LIN {X -0.181,Y -423.793,Z 1219.594,A 0.000,B 0.000,C 90.000,E1 286.913} C_DIS
LIN {X -0.003,Y -430.915,Z 1219.589,A 0.000,B 0.000,C 90.000,E1 286.079} C_DIS
LIN {X -0.077,Y -435.410,Z 1219.586,A 0.000,B 0.000,C 90.000,E1 285.552} C_DIS
LIN {X 0.192,Y -441.538,Z 1219.582,A 0.000,B 0.000,C 90.000,E1 284.717} C_DIS
LIN {X 0.092,Y -447.112,Z 1219.578,A 0.000,B 0.000,C 90.000,E1 283.939} C_DIS
LIN {X -0.076,Y -452.101,Z 1219.573,A 0.000,B 0.000,C 90.000,E1 283.175} C_DIS
LIN {X 0.247,Y -456.380,Z 1219.569,A 0.000,B 0.000,C 90.000,E1 282.355} C_DIS
LIN {X 0.160,Y -459.934,Z 1219.564,A 0.000,B 0.000,C 90.000,E1 281.591} C_DIS
LIN {X 0.182,Y -461.942,Z 1219.562,A 0.000,B 0.000,C 90.000,E1 281.074} C_DIS
LIN {X -0.154,Y -463.736,Z 1219.559,A 0.000,B 0.000,C 90.000,E1 280.602} C_DIS
LIN {X -0.028,Y -465.195,Z 1219.556,A 0.000,B 0.000,C 90.000,E1 280.074} C_DIS
LIN {X 0.030,Y -466.423,Z 1219.553,A 0.000,B 0.000,C 90.000,E1 279.557} C_DIS
LIN {X 0.174,Y -467.373,Z 1219.550,A 0.000,B 0.000,C 90.000,E1 279.029} C_DIS
LIN {X -0.212,Y -468.042,Z 1219.547,A 0.000,B 0.000,C 90.000,E1 278.568} C_DIS
LIN {X -0.128,Y -468.455,Z 1219.545,A 0.000,B 0.000,C 90.000,E1 278.049} C_DIS
LIN {X -0.038,Y -468.559,Z 1219.542,A 0.000,B 0.000,C 90.000,E1 277.530} C_DIS
LIN {X 0.114,Y -468.268,Z 1219.539,A 0.000,B 0.000,C 90.000,E1 277.004} C_DIS
LIN {X 0.206,Y -467.592,Z 1219.536,A 0.000,B 0.000,C 90.000,E1 276.486} C_DIS
LIN {X -0.168,Y -466.535,Z 1219.533,A 0.000,B 0.000,C 90.000,E1 276.024} C_DIS
LIN {X -0.127,Y -465.025,Z 1219.531,A 0.000,B 0.000,C 90.000,E1 275.511} C_DIS
LIN {X 0.240,Y -461.969,Z 1219.526,A 0.000,B 0.000,C 90.000,E1 274.702} C_DIS
LIN {X -0.194,Y -459.223,Z 1219.523,A 0.000,B 0.000,C 90.000,E1 274.245} C_DIS
LIN {X -0.149,Y -455.714,Z 1219.521,A 0.000,B 0.000,C 90.000,E1 273.726} C_DIS
LIN {X -0.151,Y -451.325,Z 1219.518,A 0.000,B 0.000,C 90.000,E1 273.212} C_DIS
LIN {X -0.063,Y -445.903,Z 1219.515,A 0.000,B 0.000,C 90.000,E1 272.694} C_DIS
LIN {X -0.214,Y -442.714,Z 1219.514,A 0.000,B 0.000,C 90.000,E1 272.465} C_DIS
LIN {X 0.026,Y -436.059,Z 1219.511,A 0.000,B 0.000,C 90.000,E1 272.007} C_DIS
LIN {X -0.048,Y -428.864,Z 1219.509,A 0.000,B 0.000,C 90.000,E1 271.661} C_DIS
LIN {X -0.016,Y -421.713,Z 1219.508,A 0.000,B 0.000,C 90.000,E1 271.375} C_DIS
LIN {X 0.042,Y -411.638,Z 1219.506,A 0.000,B 0.000,C 90.000,E1 271.031} C_DIS
LIN {X 0.082,Y -401.252,Z 1219.504,A 0.000,B 0.000,C 90.000,E1 270.745} C_DIS
LIN {X 0.155,Y -394.190,Z 1219.503,A 0.000,B 0.000,C 90.000,E1 270.573} C_DIS
LIN {X -0.024,Y -385.825,Z 1219.503,A 0.000,B 0.000,C 90.000,E1 270.458} C_DIS
LIN {X 0.033,Y -376.005,Z 1219.502,A 0.000,B 0.000,C 90.000,E1 270.344} C_DIS
LIN {X 0.010,Y -364.057,Z 1219.502,A 0.000,B 0.000,C 90.000,E1 270.286} C_DIS
LIN {X -0.027,Y -181.581,Z 1219.502,A 0.000,B 0.000,C 90.000,E1 270.286} C_DIS
LIN {X -0.048,Y -180.830,Z 1219.472,A 0.000,B 0.000,C 90.000,E1 264.894} C_DIS
LIN {X 0.032,Y -178.936,Z 1219.443,A 0.000,B 0.000,C 90.000,E1 259.803} C_DIS
LIN {X -0.100,Y -175.984,Z 1219.415,A 0.000,B 0.000,C 90.000,E1 254.755} C_DIS
LIN {X 0.015,Y -175.481,Z 1219.410,A 0.000,B 0.000,C 90.000,E1 253.866} C_DIS
LIN {X 0.072,Y -172.227,Z 1219.387,A 0.000,B 0.000,C 90.000,E1 249.571} C_DIS
LIN {X 0.049,Y -171.704,Z 1219.382,A 0.000,B 0.000,C 90.000,E1 248.720} C_DIS
LIN {X -0.026,Y -167.298,Z 1219.353,A 0.000,B 0.000,C 90.000,E1 243.563} C_DIS
LIN {X 0.056,Y -166.676,Z 1219.348,A 0.000,B 0.000,C 90.000,E1 242.666} C_DIS
LIN {X -0.029,Y -162.658,Z 1219.324,A 0.000,B 0.000,C 90.000,E1 238.329} C_DIS
LIN {X 0.033,Y -161.347,Z 1219.314,A 0.000,B 0.000,C 90.000,E1 236.548} C_DIS
LIN {X 0.076,Y -157.341,Z 1219.290,A 0.000,B 0.000,C 90.000,E1 232.110} C_DIS
LIN {X 0.008,Y -155.327,Z 1219.275,A 0.000,B 0.000,C 90.000,E1 229.461} C_DIS
LIN {X -0.062,Y -151.679,Z 1219.250,A 0.000,B 0.000,C 90.000,E1 225.000} C_DIS
LIN {X -0.014,Y -150.543,Z 1219.240,A 0.000,B 0.000,C 90.000,E1 223.176} C_DIS
LIN {X 0.020,Y -147.269,Z 1219.215,A 0.000,B 0.000,C 90.000,E1 218.624} C_DIS
LIN {X -0.007,Y -145.296,Z 1219.194,A 0.000,B 0.000,C 90.000,E1 214.978} C_DIS
LIN {X -0.015,Y -142.392,Z 1219.164,A 0.000,B 0.000,C 90.000,E1 209.461} C_DIS
LIN {X 0.031,Y -141.372,Z 1219.148,A 0.000,B 0.000,C 90.000,E1 206.668} C_DIS
LIN {X 0.009,Y -139.346,Z 1219.112,A 0.000,B 0.000,C 90.000,E1 200.174} C_DIS
LIN {X 0.014,Y -139.018,Z 1219.102,A 0.000,B 0.000,C 90.000,E1 198.308} C_DIS
LIN {X 0.010,Y -138.343,Z 1219.055,A 0.000,B 0.000,C 90.000,E1 189.905} C_DIS
LIN {X 0.030,Y -139.392,Z 1219.008,A 0.000,B 0.000,C 90.000,E1 181.489} C_DIS
LIN {X -0.057,Y -141.291,Z 1218.972,A 0.000,B 0.000,C 90.000,E1 175.008} C_DIS
LIN {X 0.042,Y -142.654,Z 1218.957,A 0.000,B 0.000,C 90.000,E1 172.186} C_DIS
LIN {X -0.008,Y -144.994,Z 1218.931,A 0.000,B 0.000,C 90.000,E1 167.589} C_DIS
LIN {X -0.019,Y -147.621,Z 1218.911,A 0.000,B 0.000,C 90.000,E1 163.921} C_DIS
LIN {X 0.060,Y -150.248,Z 1218.890,A 0.000,B 0.000,C 90.000,E1 160.242} C_DIS
LIN {X -0.067,Y -153.643,Z 1218.870,A 0.000,B 0.000,C 90.000,E1 156.666} C_DIS
LIN {X -0.009,Y -157.059,Z 1218.850,A 0.000,B 0.000,C 90.000,E1 153.050} C_DIS
LIN {X 0.071,Y -161.189,Z 1218.830,A 0.000,B 0.000,C 90.000,E1 149.459} C_DIS
LIN {X 0.019,Y -163.281,Z 1218.821,A 0.000,B 0.000,C 90.000,E1 147.709} C_DIS
LIN {X 0.029,Y -167.725,Z 1218.801,A 0.000,B 0.000,C 90.000,E1 144.196} C_DIS
LIN {X -0.058,Y -171.543,Z 1218.787,A 0.000,B 0.000,C 90.000,E1 141.618} C_DIS
LIN {X -0.016,Y -176.486,Z 1218.768,A 0.000,B 0.000,C 90.000,E1 138.162} C_DIS
LIN {X 0.109,Y -180.783,Z 1218.753,A 0.000,B 0.000,C 90.000,E1 135.567} C_DIS
LIN {X -0.029,Y -186.190,Z 1218.735,A 0.000,B 0.000,C 90.000,E1 132.243} C_DIS
LIN {X 0.035,Y -190.827,Z 1218.721,A 0.000,B 0.000,C 90.000,E1 129.725} C_DIS
LIN {X -0.047,Y -196.587,Z 1218.703,A 0.000,B 0.000,C 90.000,E1 126.457} C_DIS
LIN {X -0.025,Y -201.169,Z 1218.689,A 0.000,B 0.000,C 90.000,E1 124.119} C_DIS
LIN {X -0.074,Y -311.194,Z 1218.689,A 0.000,B 0.000,C 90.000,E1 124.119} C_DIS
LIN {X 0.059,Y -315.121,Z 1218.689,A 0.000,B 0.000,C 90.000,E1 123.992} C_DIS
LIN {X -0.077,Y -318.182,Z 1218.688,A 0.000,B 0.000,C 90.000,E1 123.833} C_DIS
LIN {X 0.020,Y -321.861,Z 1218.686,A 0.000,B 0.000,C 90.000,E1 123.452} C_DIS
LIN {X 0.120,Y -325.351,Z 1218.683,A 0.000,B 0.000,C 90.000,E1 122.880} C_DIS
LIN {X -0.066,Y -326.752,Z 1218.681,A 0.000,B 0.000,C 90.000,E1 122.594} C_DIS
LIN {X -0.100,Y -338.790,Z 1218.664,A 0.000,B 0.000,C 90.000,E1 119.461} C_DIS
LIN {X 0.052,Y -351.056,Z 1218.648,A 0.000,B 0.000,C 90.000,E1 116.668} C_DIS
LIN {X 0.100,Y -364.803,Z 1218.633,A 0.000,B 0.000,C 90.000,E1 113.951} C_DIS
LIN {X 0.137,Y -378.369,Z 1218.620,A 0.000,B 0.000,C 90.000,E1 111.589} C_DIS
LIN {X -0.128,Y -393.300,Z 1218.607,A 0.000,B 0.000,C 90.000,E1 109.322} C_DIS
LIN {X 0.091,Y -409.699,Z 1218.595,A 0.000,B 0.000,C 90.000,E1 107.040} C_DIS
LIN {X 0.218,Y -427.684,Z 1218.583,A 0.000,B 0.000,C 90.000,E1 104.828} C_DIS
LIN {X 0.171,Y -447.227,Z 1218.571,A 0.000,B 0.000,C 90.000,E1 102.715} C_DIS
LIN {X -0.035,Y -467.496,Z 1218.560,A 0.000,B 0.000,C 90.000,E1 100.782} C_DIS
LIN {X 0.023,Y -472.557,Z 1218.557,A 0.000,B 0.000,C 90.000,E1 100.310} C_DIS
LIN {X 0.071,Y -474.485,Z 1218.556,A 0.000,B 0.000,C 90.000,E1 100.074} C_DIS
LIN {X -0.149,Y -476.087,Z 1218.555,A 0.000,B 0.000,C 90.000,E1 99.849} C_DIS
LIN {X 0.183,Y -477.288,Z 1218.553,A 0.000,B 0.000,C 90.000,E1 99.557} C_DIS
LIN {X -0.154,Y -478.748,Z 1218.550,A 0.000,B 0.000,C 90.000,E1 99.095} C_DIS
LIN {X 0.062,Y -479.170,Z 1218.548,A 0.000,B 0.000,C 90.000,E1 98.568} C_DIS
LIN {X 0.214,Y -478.622,Z 1218.545,A 0.000,B 0.000,C 90.000,E1 98.049} C_DIS
LIN {X -0.103,Y -477.019,Z 1218.542,A 0.000,B 0.000,C 90.000,E1 97.587} C_DIS
LIN {X 0.241,Y -475.734,Z 1218.541,A 0.000,B 0.000,C 90.000,E1 97.296} C_DIS
LIN {X 0.187,Y -470.283,Z 1218.536,A 0.000,B 0.000,C 90.000,E1 96.549} C_DIS
LIN {X -0.178,Y -454.020,Z 1218.524,A 0.000,B 0.000,C 90.000,E1 94.302} C_DIS
LIN {X 0.078,Y -436.846,Z 1218.509,A 0.000,B 0.000,C 90.000,E1 91.661} C_DIS
LIN {X -0.022,Y -424.151,Z 1218.497,A 0.000,B 0.000,C 90.000,E1 89.542} C_DIS
LIN {X 0.110,Y -410.868,Z 1218.484,A 0.000,B 0.000,C 90.000,E1 87.078} C_DIS
LIN {X -0.112,Y -399.375,Z 1218.472,A 0.000,B 0.000,C 90.000,E1 84.894} C_DIS
LIN {X -0.169,Y -389.148,Z 1218.461,A 0.000,B 0.000,C 90.000,E1 82.932} C_DIS
LIN {X 0.002,Y -378.897,Z 1218.449,A 0.000,B 0.000,C 90.000,E1 80.905} C_DIS
LIN {X 0.010,Y -369.792,Z 1218.440,A 0.000,B 0.000,C 90.000,E1 79.162} C_DIS
LIN {X -0.082,Y -360.382,Z 1218.430,A 0.000,B 0.000,C 90.000,E1 77.409} C_DIS
LIN {X 0.099,Y -349.180,Z 1218.418,A 0.000,B 0.000,C 90.000,E1 75.283} C_DIS
LIN {X 0.130,Y -337.941,Z 1218.406,A 0.000,B 0.000,C 90.000,E1 73.142} C_DIS
LIN {X -0.025,Y -325.335,Z 1218.393,A 0.000,B 0.000,C 90.000,E1 70.678} C_DIS
LIN {X -0.098,Y -308.752,Z 1218.373,A 0.000,B 0.000,C 90.000,E1 67.177} C_DIS
LIN {X -0.096,Y -294.911,Z 1218.355,A 0.000,B 0.000,C 90.000,E1 63.896} C_DIS
LIN {X 0.015,Y -282.061,Z 1218.336,A 0.000,B 0.000,C 90.000,E1 60.511} C_DIS
LIN {X 0.143,Y -270.174,Z 1218.317,A 0.000,B 0.000,C 90.000,E1 57.041} C_DIS
LIN {X -0.002,Y -260.275,Z 1218.299,A 0.000,B 0.000,C 90.000,E1 53.909} C_DIS
LIN {X 0.030,Y -252.023,Z 1218.284,A 0.000,B 0.000,C 90.000,E1 51.045} C_DIS
LIN {X 0.103,Y -242.407,Z 1218.263,A 0.000,B 0.000,C 90.000,E1 47.391} C_DIS
LIN {X 0.021,Y -233.243,Z 1218.243,A 0.000,B 0.000,C 90.000,E1 43.704} C_DIS
LIN {X -0.028,Y -226.234,Z 1218.226,A 0.000,B 0.000,C 90.000,E1 40.701} C_DIS
LIN {X -0.025,Y -217.990,Z 1218.205,A 0.000,B 0.000,C 90.000,E1 36.870} C_DIS
LIN {X -0.125,Y -212.135,Z 1218.188,A 0.000,B 0.000,C 90.000,E1 33.785} C_DIS
LIN {X 0.048,Y -205.769,Z 1218.166,A 0.000,B 0.000,C 90.000,E1 29.795} C_DIS
LIN {X 0.054,Y -200.364,Z 1218.143,A 0.000,B 0.000,C 90.000,E1 25.796} C_DIS
LIN {X -0.002,Y -195.781,Z 1218.121,A 0.000,B 0.000,C 90.000,E1 21.770} C_DIS
LIN {X -0.020,Y -191.988,Z 1218.098,A 0.000,B 0.000,C 90.000,E1 17.692} C_DIS
LIN {X -0.089,Y -188.597,Z 1218.071,A 0.000,B 0.000,C 90.000,E1 12.771} C_DIS
LIN {X 0.054,Y -186.067,Z 1218.034,A 0.000,B 0.000,C 90.000,E1 6.087} C_DIS
LIN {X 0.041,Y -187.339,Z 1217.974,A 0.000,B 0.000,C 90.000,E1 355.355} C_DIS
LIN {X -0.010,Y -190.596,Z 1217.942,A 0.000,B 0.000,C 90.000,E1 349.567} C_DIS
LIN {X -0.006,Y -194.831,Z 1217.915,A 0.000,B 0.000,C 90.000,E1 344.629} C_DIS
LIN {X 0.004,Y -199.290,Z 1217.892,A 0.000,B 0.000,C 90.000,E1 340.550} C_DIS
LIN {X -0.076,Y -204.530,Z 1217.870,A 0.000,B 0.000,C 90.000,E1 336.538} C_DIS
LIN {X -0.032,Y -210.424,Z 1217.847,A 0.000,B 0.000,C 90.000,E1 332.538} C_DIS
LIN {X 0.033,Y -216.721,Z 1217.826,A 0.000,B 0.000,C 90.000,E1 328.584} C_DIS
LIN {X 0.083,Y -223.667,Z 1217.804,A 0.000,B 0.000,C 90.000,E1 324.689} C_DIS
LIN {X 0.002,Y -231.308,Z 1217.783,A 0.000,B 0.000,C 90.000,E1 320.884} C_DIS
LIN {X -0.116,Y -239.837,Z 1217.762,A 0.000,B 0.000,C 90.000,E1 317.148} C_DIS
LIN {X 0.032,Y -248.751,Z 1217.743,A 0.000,B 0.000,C 90.000,E1 313.785} C_DIS
LIN {X 0.084,Y -256.811,Z 1217.729,A 0.000,B 0.000,C 90.000,E1 311.229} C_DIS
LIN {X 0.109,Y -268.692,Z 1217.711,A 0.000,B 0.000,C 90.000,E1 308.016} C_DIS
LIN {X -0.045,Y -275.951,Z 1217.702,A 0.000,B 0.000,C 90.000,E1 306.297} C_DIS
LIN {X 0.188,Y -288.819,Z 1217.686,A 0.000,B 0.000,C 90.000,E1 303.499} C_DIS
LIN {X -0.099,Y -304.915,Z 1217.670,A 0.000,B 0.000,C 90.000,E1 300.541} C_DIS
LIN {X -0.013,Y -310.756,Z 1217.664,A 0.000,B 0.000,C 90.000,E1 299.539} C_DIS
LIN {X -0.017,Y -317.538,Z 1217.659,A 0.000,B 0.000,C 90.000,E1 298.565} C_DIS
LIN {X -0.057,Y -334.956,Z 1217.646,A 0.000,B 0.000,C 90.000,E1 296.360} C_DIS
LIN {X 0.162,Y -350.706,Z 1217.636,A 0.000,B 0.000,C 90.000,E1 294.515} C_DIS
LIN {X 0.188,Y -372.016,Z 1217.624,A 0.000,B 0.000,C 90.000,E1 292.206} C_DIS
LIN {X -0.160,Y -387.910,Z 1217.614,A 0.000,B 0.000,C 90.000,E1 290.610} C_DIS
LIN {X 0.093,Y -403.621,Z 1217.605,A 0.000,B 0.000,C 90.000,E1 288.960} C_DIS
LIN {X -0.091,Y -414.002,Z 1217.599,A 0.000,B 0.000,C 90.000,E1 287.928} C_DIS
LIN {X 0.040,Y -423.975,Z 1217.594,A 0.000,B 0.000,C 90.000,E1 286.858} C_DIS
LIN {X -0.197,Y -431.096,Z 1217.589,A 0.000,B 0.000,C 90.000,E1 286.079} C_DIS
LIN {X 0.026,Y -437.688,Z 1217.585,A 0.000,B 0.000,C 90.000,E1 285.245} C_DIS
LIN {X -0.220,Y -443.611,Z 1217.580,A 0.000,B 0.000,C 90.000,E1 284.481} C_DIS
LIN {X 0.123,Y -449.018,Z 1217.576,A 0.000,B 0.000,C 90.000,E1 283.647} C_DIS
LIN {X -0.024,Y -453.766,Z 1217.572,A 0.000,B 0.000,C 90.000,E1 282.883} C_DIS
LIN {X -0.134,Y -457.773,Z 1217.567,A 0.000,B 0.000,C 90.000,E1 282.119} C_DIS
LIN {X -0.039,Y -460.049,Z 1217.564,A 0.000,B 0.000,C 90.000,E1 281.591} C_DIS
LIN {X -0.017,Y -462.068,Z 1217.562,A 0.000,B 0.000,C 90.000,E1 281.074} C_DIS
LIN {X 0.103,Y -463.857,Z 1217.559,A 0.000,B 0.000,C 90.000,E1 280.546} C_DIS
LIN {X 0.231,Y -465.337,Z 1217.556,A 0.000,B 0.000,C 90.000,E1 280.018} C_DIS
LIN {X -0.169,Y -466.544,Z 1217.553,A 0.000,B 0.000,C 90.000,E1 279.557} C_DIS
LIN {X -0.026,Y -467.468,Z 1217.550,A 0.000,B 0.000,C 90.000,E1 279.029} C_DIS
LIN {X 0.052,Y -468.138,Z 1217.547,A 0.000,B 0.000,C 90.000,E1 278.511} C_DIS
LIN {X 0.138,Y -468.547,Z 1217.545,A 0.000,B 0.000,C 90.000,E1 277.992} C_DIS
LIN {X -0.235,Y -468.647,Z 1217.542,A 0.000,B 0.000,C 90.000,E1 277.530} C_DIS
LIN {X -0.082,Y -468.386,Z 1217.539,A 0.000,B 0.000,C 90.000,E1 277.004} C_DIS
LIN {X 0.010,Y -467.717,Z 1217.536,A 0.000,B 0.000,C 90.000,E1 276.486} C_DIS
LIN {X 0.101,Y -466.635,Z 1217.533,A 0.000,B 0.000,C 90.000,E1 275.967} C_DIS
LIN {X 0.143,Y -465.168,Z 1217.530,A 0.000,B 0.000,C 90.000,E1 275.454} C_DIS
LIN {X -0.237,Y -463.243,Z 1217.528,A 0.000,B 0.000,C 90.000,E1 274.992} C_DIS
LIN {X -0.164,Y -460.800,Z 1217.525,A 0.000,B 0.000,C 90.000,E1 274.473} C_DIS
LIN {X -0.112,Y -457.674,Z 1217.522,A 0.000,B 0.000,C 90.000,E1 273.955} C_DIS
LIN {X 0.118,Y -455.850,Z 1217.521,A 0.000,B 0.000,C 90.000,E1 273.669} C_DIS
LIN {X 0.114,Y -451.401,Z 1217.518,A 0.000,B 0.000,C 90.000,E1 273.154} C_DIS
LIN {X -0.092,Y -448.802,Z 1217.516,A 0.000,B 0.000,C 90.000,E1 272.922} C_DIS
LIN {X 0.016,Y -442.633,Z 1217.513,A 0.000,B 0.000,C 90.000,E1 272.407} C_DIS
LIN {X -0.151,Y -436.063,Z 1217.511,A 0.000,B 0.000,C 90.000,E1 272.007} C_DIS
LIN {X 0.215,Y -428.691,Z 1217.509,A 0.000,B 0.000,C 90.000,E1 271.604} C_DIS
LIN {X -0.117,Y -421.712,Z 1217.508,A 0.000,B 0.000,C 90.000,E1 271.375} C_DIS
LIN {X -0.035,Y -411.626,Z 1217.506,A 0.000,B 0.000,C 90.000,E1 271.031} C_DIS
LIN {X -0.029,Y -401.197,Z 1217.504,A 0.000,B 0.000,C 90.000,E1 270.745} C_DIS
LIN {X 0.041,Y -394.037,Z 1217.503,A 0.000,B 0.000,C 90.000,E1 270.573} C_DIS
LIN {X -0.126,Y -385.717,Z 1217.502,A 0.000,B 0.000,C 90.000,E1 270.458} C_DIS
LIN {X -0.054,Y -376.259,Z 1217.502,A 0.000,B 0.000,C 90.000,E1 270.344} C_DIS
LIN {X -0.078,Y -364.203,Z 1217.501,A 0.000,B 0.000,C 90.000,E1 270.286} C_DIS
LIN {X -0.072,Y -181.581,Z 1217.501,A 0.000,B 0.000,C 90.000,E1 270.286} C_DIS
LIN {X 0.088,Y -180.826,Z 1217.471,A 0.000,B 0.000,C 90.000,E1 264.837} C_DIS
LIN {X -0.012,Y -178.930,Z 1217.443,A 0.000,B 0.000,C 90.000,E1 259.803} C_DIS
LIN {X 0.026,Y -175.979,Z 1217.415,A 0.000,B 0.000,C 90.000,E1 254.700} C_DIS
LIN {X -0.030,Y -175.468,Z 1217.410,A 0.000,B 0.000,C 90.000,E1 253.866} C_DIS
LIN {X 0.028,Y -172.218,Z 1217.387,A 0.000,B 0.000,C 90.000,E1 249.571} C_DIS
LIN {X 0.005,Y -171.694,Z 1217.382,A 0.000,B 0.000,C 90.000,E1 248.720} C_DIS
LIN {X 0.081,Y -167.288,Z 1217.353,A 0.000,B 0.000,C 90.000,E1 243.512} C_DIS
LIN {X 0.014,Y -166.664,Z 1217.348,A 0.000,B 0.000,C 90.000,E1 242.666} C_DIS
LIN {X -0.071,Y -162.646,Z 1217.324,A 0.000,B 0.000,C 90.000,E1 238.329} C_DIS
LIN {X -0.008,Y -161.335,Z 1217.314,A 0.000,B 0.000,C 90.000,E1 236.548} C_DIS
LIN {X 0.035,Y -157.331,Z 1217.290,A 0.000,B 0.000,C 90.000,E1 232.110} C_DIS
LIN {X -0.032,Y -155.313,Z 1217.275,A 0.000,B 0.000,C 90.000,E1 229.461} C_DIS
LIN {X 0.005,Y -151.669,Z 1217.250,A 0.000,B 0.000,C 90.000,E1 224.960} C_DIS
LIN {X -0.053,Y -150.535,Z 1217.240,A 0.000,B 0.000,C 90.000,E1 223.176} C_DIS
LIN {X -0.020,Y -147.259,Z 1217.214,A 0.000,B 0.000,C 90.000,E1 218.624} C_DIS
LIN {X 0.037,Y -145.286,Z 1217.194,A 0.000,B 0.000,C 90.000,E1 214.945} C_DIS
LIN {X 0.071,Y -142.386,Z 1217.164,A 0.000,B 0.000,C 90.000,E1 209.411} C_DIS
LIN {X -0.007,Y -141.364,Z 1217.148,A 0.000,B 0.000,C 90.000,E1 206.668} C_DIS
LIN {X -0.029,Y -139.344,Z 1217.112,A 0.000,B 0.000,C 90.000,E1 200.174} C_DIS
LIN {X -0.024,Y -139.014,Z 1217.102,A 0.000,B 0.000,C 90.000,E1 198.308} C_DIS
LIN {X -0.028,Y -138.341,Z 1217.055,A 0.000,B 0.000,C 90.000,E1 189.905} C_DIS
LIN {X -0.008,Y -139.397,Z 1217.008,A 0.000,B 0.000,C 90.000,E1 181.489} C_DIS
LIN {X 0.045,Y -141.298,Z 1216.972,A 0.000,B 0.000,C 90.000,E1 174.951} C_DIS
LIN {X 0.003,Y -142.660,Z 1216.957,A 0.000,B 0.000,C 90.000,E1 172.186} C_DIS
LIN {X -0.047,Y -145.004,Z 1216.931,A 0.000,B 0.000,C 90.000,E1 167.589} C_DIS
LIN {X -0.058,Y -147.632,Z 1216.911,A 0.000,B 0.000,C 90.000,E1 163.921} C_DIS
LIN {X 0.020,Y -150.260,Z 1216.890,A 0.000,B 0.000,C 90.000,E1 160.242} C_DIS
LIN {X 0.033,Y -153.659,Z 1216.870,A 0.000,B 0.000,C 90.000,E1 156.613} C_DIS
LIN {X -0.050,Y -157.074,Z 1216.850,A 0.000,B 0.000,C 90.000,E1 153.050} C_DIS
LIN {X 0.029,Y -161.208,Z 1216.830,A 0.000,B 0.000,C 90.000,E1 149.459} C_DIS
LIN {X -0.024,Y -163.298,Z 1216.821,A 0.000,B 0.000,C 90.000,E1 147.709} C_DIS
LIN {X -0.013,Y -167.745,Z 1216.801,A 0.000,B 0.000,C 90.000,E1 144.196} C_DIS
LIN {X -0.101,Y -171.562,Z 1216.787,A 0.000,B 0.000,C 90.000,E1 141.618} C_DIS
LIN {X -0.060,Y -176.508,Z 1216.767,A 0.000,B 0.000,C 90.000,E1 138.162} C_DIS
LIN {X 0.065,Y -180.806,Z 1216.753,A 0.000,B 0.000,C 90.000,E1 135.567} C_DIS
LIN {X 0.051,Y -186.214,Z 1216.734,A 0.000,B 0.000,C 90.000,E1 132.204} C_DIS
LIN {X -0.011,Y -190.851,Z 1216.721,A 0.000,B 0.000,C 90.000,E1 129.725} C_DIS
LIN {X 0.023,Y -196.613,Z 1216.702,A 0.000,B 0.000,C 90.000,E1 126.423} C_DIS
LIN {X -0.030,Y -201.171,Z 1216.689,A 0.000,B 0.000,C 90.000,E1 124.119} C_DIS
LIN {X 0.046,Y -201.214,Z 1216.689,A 0.000,B 0.000,C 90.000,E1 124.072} C_DIS
LIN {X 0.035,Y -311.295,Z 1216.689,A 0.000,B 0.000,C 90.000,E1 124.072} C_DIS
LIN {X -0.071,Y -312.635,Z 1216.689,A 0.000,B 0.000,C 90.000,E1 124.072} C_DIS
LIN {X -0.016,Y -314.876,Z 1216.689,A 0.000,B 0.000,C 90.000,E1 123.992} C_DIS
LIN {X 0.044,Y -318.236,Z 1216.688,A 0.000,B 0.000,C 90.000,E1 123.785} C_DIS
LIN {X -0.074,Y -321.847,Z 1216.686,A 0.000,B 0.000,C 90.000,E1 123.452} C_DIS
LIN {X 0.044,Y -325.356,Z 1216.683,A 0.000,B 0.000,C 90.000,E1 122.880} C_DIS
LIN {X 0.133,Y -326.774,Z 1216.681,A 0.000,B 0.000,C 90.000,E1 122.546} C_DIS
LIN {X 0.117,Y -338.823,Z 1216.663,A 0.000,B 0.000,C 90.000,E1 119.411} C_DIS
LIN {X -0.028,Y -351.096,Z 1216.648,A 0.000,B 0.000,C 90.000,E1 116.668} C_DIS
LIN {X 0.017,Y -364.851,Z 1216.633,A 0.000,B 0.000,C 90.000,E1 113.951} C_DIS
LIN {X 0.052,Y -378.424,Z 1216.620,A 0.000,B 0.000,C 90.000,E1 111.589} C_DIS
LIN {X 0.157,Y -393.362,Z 1216.607,A 0.000,B 0.000,C 90.000,E1 109.268} C_DIS
LIN {X 0.003,Y -409.769,Z 1216.595,A 0.000,B 0.000,C 90.000,E1 107.040} C_DIS
LIN {X 0.128,Y -427.762,Z 1216.583,A 0.000,B 0.000,C 90.000,E1 104.828} C_DIS
LIN {X 0.082,Y -447.311,Z 1216.571,A 0.000,B 0.000,C 90.000,E1 102.715} C_DIS
LIN {X -0.122,Y -467.582,Z 1216.560,A 0.000,B 0.000,C 90.000,E1 100.782} C_DIS
LIN {X -0.063,Y -472.613,Z 1216.557,A 0.000,B 0.000,C 90.000,E1 100.310} C_DIS
LIN {X -0.014,Y -474.496,Z 1216.556,A 0.000,B 0.000,C 90.000,E1 100.074} C_DIS
LIN {X -0.235,Y -476.063,Z 1216.555,A 0.000,B 0.000,C 90.000,E1 99.849} C_DIS
LIN {X 0.096,Y -477.237,Z 1216.553,A 0.000,B 0.000,C 90.000,E1 99.557} C_DIS
LIN {X -0.165,Y -478.657,Z 1216.550,A 0.000,B 0.000,C 90.000,E1 99.086} C_DIS
LIN {X -0.025,Y -479.042,Z 1216.548,A 0.000,B 0.000,C 90.000,E1 98.568} C_DIS
LIN {X 0.127,Y -478.457,Z 1216.545,A 0.000,B 0.000,C 90.000,E1 98.049} C_DIS
LIN {X -0.190,Y -476.811,Z 1216.542,A 0.000,B 0.000,C 90.000,E1 97.587} C_DIS
LIN {X 0.153,Y -475.500,Z 1216.541,A 0.000,B 0.000,C 90.000,E1 97.296} C_DIS
LIN {X -0.158,Y -462.766,Z 1216.531,A 0.000,B 0.000,C 90.000,E1 95.568} C_DIS
LIN {X -0.123,Y -441.667,Z 1216.514,A 0.000,B 0.000,C 90.000,E1 92.465} C_DIS
LIN {X 0.040,Y -426.995,Z 1216.500,A 0.000,B 0.000,C 90.000,E1 90.057} C_DIS
LIN {X -0.076,Y -412.105,Z 1216.485,A 0.000,B 0.000,C 90.000,E1 87.364} C_DIS
LIN {X 0.139,Y -400.613,Z 1216.473,A 0.000,B 0.000,C 90.000,E1 85.122} C_DIS
LIN {X 0.063,Y -390.406,Z 1216.462,A 0.000,B 0.000,C 90.000,E1 83.166} C_DIS
LIN {X -0.132,Y -380.151,Z 1216.451,A 0.000,B 0.000,C 90.000,E1 81.197} C_DIS
LIN {X -0.103,Y -372.647,Z 1216.443,A 0.000,B 0.000,C 90.000,E1 79.746} C_DIS
LIN {X -0.140,Y -363.311,Z 1216.433,A 0.000,B 0.000,C 90.000,E1 77.993} C_DIS
LIN {X 0.080,Y -353.756,Z 1216.423,A 0.000,B 0.000,C 90.000,E1 76.172} C_DIS
LIN {X 0.110,Y -342.546,Z 1216.411,A 0.000,B 0.000,C 90.000,E1 74.047} C_DIS
LIN {X 0.060,Y -329.810,Z 1216.398,A 0.000,B 0.000,C 90.000,E1 71.583} C_DIS
LIN {X -0.133,Y -315.908,Z 1216.382,A 0.000,B 0.000,C 90.000,E1 68.773} C_DIS
LIN {X 0.009,Y -300.112,Z 1216.362,A 0.000,B 0.000,C 90.000,E1 65.177} C_DIS
LIN {X -0.002,Y -286.902,Z 1216.344,A 0.000,B 0.000,C 90.000,E1 61.847} C_DIS
LIN {X -0.109,Y -274.583,Z 1216.325,A 0.000,B 0.000,C 90.000,E1 58.456} C_DIS
LIN {X -0.058,Y -264.361,Z 1216.307,A 0.000,B 0.000,C 90.000,E1 55.308} C_DIS
LIN {X 0.002,Y -253.798,Z 1216.287,A 0.000,B 0.000,C 90.000,E1 51.743} C_DIS
LIN {X 0.001,Y -243.978,Z 1216.267,A 0.000,B 0.000,C 90.000,E1 48.119} C_DIS
LIN {X 0.029,Y -236.496,Z 1216.251,A 0.000,B 0.000,C 90.000,E1 45.162} C_DIS
LIN {X 0.048,Y -229.348,Z 1216.234,A 0.000,B 0.000,C 90.000,E1 42.162} C_DIS
LIN {X -0.057,Y -220.795,Z 1216.213,A 0.000,B 0.000,C 90.000,E1 38.382} C_DIS
LIN {X 0.036,Y -214.593,Z 1216.196,A 0.000,B 0.000,C 90.000,E1 35.264} C_DIS
LIN {X 0.049,Y -207.862,Z 1216.174,A 0.000,B 0.000,C 90.000,E1 31.337} C_DIS
LIN {X -0.048,Y -202.119,Z 1216.152,A 0.000,B 0.000,C 90.000,E1 27.385} C_DIS
LIN {X 0.034,Y -197.219,Z 1216.130,A 0.000,B 0.000,C 90.000,E1 23.334} C_DIS
LIN {X 0.018,Y -193.068,Z 1216.107,A 0.000,B 0.000,C 90.000,E1 19.268} C_DIS
LIN {X -0.044,Y -189.241,Z 1216.080,A 0.000,B 0.000,C 90.000,E1 14.356} C_DIS
LIN {X -0.087,Y -186.414,Z 1216.047,A 0.000,B 0.000,C 90.000,E1 8.568} C_DIS
LIN {X -0.043,Y -187.379,Z 1215.970,A 0.000,B 0.000,C 90.000,E1 354.546} C_DIS
LIN {X -0.034,Y -190.265,Z 1215.942,A 0.000,B 0.000,C 90.000,E1 349.567} C_DIS
LIN {X -0.042,Y -194.537,Z 1215.915,A 0.000,B 0.000,C 90.000,E1 344.629} C_DIS
LIN {X -0.044,Y -199.016,Z 1215.892,A 0.000,B 0.000,C 90.000,E1 340.550} C_DIS
LIN {X 0.054,Y -204.282,Z 1215.870,A 0.000,B 0.000,C 90.000,E1 336.485} C_DIS
LIN {X 0.088,Y -210.174,Z 1215.847,A 0.000,B 0.000,C 90.000,E1 332.487} C_DIS
LIN {X -0.044,Y -216.505,Z 1215.825,A 0.000,B 0.000,C 90.000,E1 328.584} C_DIS
LIN {X -0.004,Y -223.450,Z 1215.804,A 0.000,B 0.000,C 90.000,E1 324.689} C_DIS
LIN {X 0.015,Y -229.521,Z 1215.787,A 0.000,B 0.000,C 90.000,E1 321.618} C_DIS
LIN {X 0.020,Y -237.878,Z 1215.766,A 0.000,B 0.000,C 90.000,E1 317.838} C_DIS
LIN {X -0.061,Y -246.508,Z 1215.747,A 0.000,B 0.000,C 90.000,E1 314.514} C_DIS
LIN {X 0.111,Y -254.320,Z 1215.733,A 0.000,B 0.000,C 90.000,E1 311.919} C_DIS
LIN {X -0.041,Y -263.258,Z 1215.719,A 0.000,B 0.000,C 90.000,E1 309.439} C_DIS
LIN {X 0.125,Y -274.426,Z 1215.703,A 0.000,B 0.000,C 90.000,E1 306.583} C_DIS
LIN {X 0.052,Y -288.806,Z 1215.686,A 0.000,B 0.000,C 90.000,E1 303.499} C_DIS
LIN {X 0.175,Y -304.936,Z 1215.669,A 0.000,B 0.000,C 90.000,E1 300.463} C_DIS
LIN {X -0.159,Y -310.828,Z 1215.664,A 0.000,B 0.000,C 90.000,E1 299.539} C_DIS
LIN {X 0.068,Y -319.692,Z 1215.657,A 0.000,B 0.000,C 90.000,E1 298.231} C_DIS
LIN {X 0.041,Y -337.343,Z 1215.645,A 0.000,B 0.000,C 90.000,E1 296.027} C_DIS
LIN {X 0.179,Y -353.178,Z 1215.635,A 0.000,B 0.000,C 90.000,E1 294.207} C_DIS
LIN {X 0.201,Y -371.779,Z 1215.624,A 0.000,B 0.000,C 90.000,E1 292.206} C_DIS
LIN {X -0.074,Y -387.625,Z 1215.614,A 0.000,B 0.000,C 90.000,E1 290.610} C_DIS
LIN {X -0.138,Y -400.315,Z 1215.607,A 0.000,B 0.000,C 90.000,E1 289.322} C_DIS
LIN {X -0.044,Y -413.195,Z 1215.600,A 0.000,B 0.000,C 90.000,E1 288.000} C_DIS
LIN {X -0.151,Y -423.007,Z 1215.594,A 0.000,B 0.000,C 90.000,E1 286.985} C_DIS
LIN {X -0.165,Y -429.987,Z 1215.590,A 0.000,B 0.000,C 90.000,E1 286.205} C_DIS
LIN {X 0.051,Y -436.657,Z 1215.585,A 0.000,B 0.000,C 90.000,E1 285.371} C_DIS
LIN {X 0.120,Y -444.590,Z 1215.580,A 0.000,B 0.000,C 90.000,E1 284.300} C_DIS
LIN {X -0.063,Y -449.897,Z 1215.575,A 0.000,B 0.000,C 90.000,E1 283.536} C_DIS
LIN {X -0.205,Y -454.519,Z 1215.571,A 0.000,B 0.000,C 90.000,E1 282.771} C_DIS
LIN {X 0.144,Y -458.416,Z 1215.567,A 0.000,B 0.000,C 90.000,E1 281.951} C_DIS
LIN {X 0.078,Y -461.656,Z 1215.562,A 0.000,B 0.000,C 90.000,E1 281.186} C_DIS
LIN {X 0.199,Y -463.461,Z 1215.559,A 0.000,B 0.000,C 90.000,E1 280.658} C_DIS
LIN {X -0.215,Y -465.019,Z 1215.557,A 0.000,B 0.000,C 90.000,E1 280.197} C_DIS
LIN {X -0.079,Y -466.313,Z 1215.554,A 0.000,B 0.000,C 90.000,E1 279.670} C_DIS
LIN {X -0.013,Y -467.322,Z 1215.551,A 0.000,B 0.000,C 90.000,E1 279.151} C_DIS
LIN {X 0.136,Y -468.073,Z 1215.548,A 0.000,B 0.000,C 90.000,E1 278.624} C_DIS
LIN {X 0.220,Y -468.533,Z 1215.545,A 0.000,B 0.000,C 90.000,E1 278.106} C_DIS
LIN {X -0.155,Y -468.739,Z 1215.542,A 0.000,B 0.000,C 90.000,E1 277.644} C_DIS
LIN {X -0.060,Y -468.594,Z 1215.540,A 0.000,B 0.000,C 90.000,E1 277.125} C_DIS
LIN {X 0.036,Y -468.044,Z 1215.537,A 0.000,B 0.000,C 90.000,E1 276.606} C_DIS
LIN {X 0.131,Y -467.108,Z 1215.534,A 0.000,B 0.000,C 90.000,E1 276.087} C_DIS
LIN {X -0.241,Y -465.782,Z 1215.531,A 0.000,B 0.000,C 90.000,E1 275.625} C_DIS
LIN {X -0.156,Y -464.006,Z 1215.528,A 0.000,B 0.000,C 90.000,E1 275.106} C_DIS
LIN {X -0.080,Y -461.718,Z 1215.525,A 0.000,B 0.000,C 90.000,E1 274.588} C_DIS
LIN {X -0.057,Y -458.808,Z 1215.523,A 0.000,B 0.000,C 90.000,E1 274.073} C_DIS
LIN {X -0.014,Y -455.130,Z 1215.520,A 0.000,B 0.000,C 90.000,E1 273.555} C_DIS
LIN {X 0.005,Y -450.448,Z 1215.517,A 0.000,B 0.000,C 90.000,E1 273.037} C_DIS
LIN {X -0.217,Y -447.689,Z 1215.516,A 0.000,B 0.000,C 90.000,E1 272.808} C_DIS
LIN {X 0.085,Y -441.488,Z 1215.513,A 0.000,B 0.000,C 90.000,E1 272.293} C_DIS
LIN {X 0.159,Y -438.098,Z 1215.512,A 0.000,B 0.000,C 90.000,E1 272.064} C_DIS
LIN {X -0.033,Y -431.005,Z 1215.510,A 0.000,B 0.000,C 90.000,E1 271.718} C_DIS
LIN {X -0.084,Y -423.790,Z 1215.508,A 0.000,B 0.000,C 90.000,E1 271.432} C_DIS
LIN {X -0.078,Y -413.723,Z 1215.506,A 0.000,B 0.000,C 90.000,E1 271.088} C_DIS
LIN {X -0.120,Y -403.469,Z 1215.504,A 0.000,B 0.000,C 90.000,E1 270.802} C_DIS
LIN {X 0.185,Y -392.927,Z 1215.503,A 0.000,B 0.000,C 90.000,E1 270.516} C_DIS
LIN {X 0.076,Y -384.532,Z 1215.502,A 0.000,B 0.000,C 90.000,E1 270.401} C_DIS
LIN {X 0.020,Y -372.129,Z 1215.502,A 0.000,B 0.000,C 90.000,E1 270.286} C_DIS
LIN {X -0.167,Y -364.329,Z 1215.501,A 0.000,B 0.000,C 90.000,E1 270.286} C_DIS
LIN {X 0.076,Y -181.581,Z 1215.501,A 0.000,B 0.000,C 90.000,E1 270.229} C_DIS
LIN {X -0.073,Y -180.890,Z 1215.473,A 0.000,B 0.000,C 90.000,E1 265.179} C_DIS
LIN {X -0.011,Y -179.014,Z 1215.445,A 0.000,B 0.000,C 90.000,E1 260.095} C_DIS
LIN {X 0.084,Y -178.639,Z 1215.440,A 0.000,B 0.000,C 90.000,E1 259.218} C_DIS
LIN {X -0.018,Y -175.690,Z 1215.412,A 0.000,B 0.000,C 90.000,E1 254.157} C_DIS
LIN {X -0.007,Y -172.406,Z 1215.388,A 0.000,B 0.000,C 90.000,E1 249.880} C_DIS
LIN {X 0.010,Y -171.219,Z 1215.379,A 0.000,B 0.000,C 90.000,E1 248.156} C_DIS
LIN {X -0.014,Y -167.502,Z 1215.355,A 0.000,B 0.000,C 90.000,E1 243.845} C_DIS
LIN {X -0.081,Y -166.898,Z 1215.350,A 0.000,B 0.000,C 90.000,E1 242.999} C_DIS
LIN {X -0.029,Y -162.205,Z 1215.321,A 0.000,B 0.000,C 90.000,E1 237.740} C_DIS
LIN {X 0.025,Y -160.779,Z 1215.311,A 0.000,B 0.000,C 90.000,E1 235.960} C_DIS
LIN {X -0.004,Y -157.572,Z 1215.291,A 0.000,B 0.000,C 90.000,E1 232.431} C_DIS
LIN {X 0.030,Y -155.603,Z 1215.276,A 0.000,B 0.000,C 90.000,E1 229.747} C_DIS
LIN {X 0.080,Y -151.883,Z 1215.251,A 0.000,B 0.000,C 90.000,E1 225.243} C_DIS
LIN {X 0.093,Y -150.110,Z 1215.236,A 0.000,B 0.000,C 90.000,E1 222.528} C_DIS
LIN {X 0.010,Y -146.906,Z 1215.211,A 0.000,B 0.000,C 90.000,E1 218.016} C_DIS
LIN {X -0.088,Y -145.492,Z 1215.196,A 0.000,B 0.000,C 90.000,E1 215.311} C_DIS
LIN {X 0.031,Y -142.899,Z 1215.170,A 0.000,B 0.000,C 90.000,E1 210.669} C_DIS
LIN {X -0.039,Y -141.520,Z 1215.150,A 0.000,B 0.000,C 90.000,E1 207.001} C_DIS
LIN {X 0.004,Y -139.395,Z 1215.114,A 0.000,B 0.000,C 90.000,E1 200.482} C_DIS
LIN {X 0.055,Y -139.106,Z 1215.103,A 0.000,B 0.000,C 90.000,E1 198.598} C_DIS
LIN {X 0.047,Y -138.353,Z 1215.057,A 0.000,B 0.000,C 90.000,E1 190.197} C_DIS
LIN {X 0.040,Y -139.511,Z 1215.005,A 0.000,B 0.000,C 90.000,E1 180.859} C_DIS
LIN {X -0.019,Y -141.157,Z 1214.974,A 0.000,B 0.000,C 90.000,E1 175.298} C_DIS
LIN {X -0.048,Y -142.536,Z 1214.958,A 0.000,B 0.000,C 90.000,E1 172.527} C_DIS
LIN {X 0.020,Y -144.806,Z 1214.933,A 0.000,B 0.000,C 90.000,E1 167.881} C_DIS
LIN {X 0.008,Y -147.426,Z 1214.912,A 0.000,B 0.000,C 90.000,E1 164.212} C_DIS
LIN {X 0.037,Y -150.003,Z 1214.892,A 0.000,B 0.000,C 90.000,E1 160.550} C_DIS
LIN {X 0.044,Y -153.334,Z 1214.872,A 0.000,B 0.000,C 90.000,E1 156.922} C_DIS
LIN {X 0.025,Y -155.869,Z 1214.857,A 0.000,B 0.000,C 90.000,E1 154.229} C_DIS
LIN {X -0.008,Y -159.722,Z 1214.837,A 0.000,B 0.000,C 90.000,E1 150.667} C_DIS
LIN {X 0.059,Y -161.961,Z 1214.827,A 0.000,B 0.000,C 90.000,E1 148.869} C_DIS
LIN {X -0.057,Y -166.152,Z 1214.808,A 0.000,B 0.000,C 90.000,E1 145.388} C_DIS
LIN {X -0.061,Y -171.165,Z 1214.788,A 0.000,B 0.000,C 90.000,E1 141.904} C_DIS
LIN {X -0.027,Y -176.044,Z 1214.769,A 0.000,B 0.000,C 90.000,E1 138.447} C_DIS
LIN {X -0.032,Y -180.300,Z 1214.755,A 0.000,B 0.000,C 90.000,E1 135.891} C_DIS
LIN {X -0.060,Y -185.711,Z 1214.736,A 0.000,B 0.000,C 90.000,E1 132.528} C_DIS
LIN {X -0.009,Y -190.318,Z 1214.722,A 0.000,B 0.000,C 90.000,E1 130.011} C_DIS
LIN {X 0.039,Y -197.644,Z 1214.699,A 0.000,B 0.000,C 90.000,E1 125.884} C_DIS
LIN {X -0.048,Y -201.261,Z 1214.689,A 0.000,B 0.000,C 90.000,E1 124.072} C_DIS
LIN {X 0.064,Y -310.941,Z 1214.689,A 0.000,B 0.000,C 90.000,E1 124.040} C_DIS
LIN {X 0.129,Y -313.289,Z 1214.689,A 0.000,B 0.000,C 90.000,E1 123.992} C_DIS
LIN {X 0.179,Y -318.649,Z 1214.687,A 0.000,B 0.000,C 90.000,E1 123.706} C_DIS
LIN {X 0.050,Y -321.502,Z 1214.686,A 0.000,B 0.000,C 90.000,E1 123.452} C_DIS
LIN {X 0.014,Y -325.156,Z 1214.683,A 0.000,B 0.000,C 90.000,E1 122.911} C_DIS
LIN {X 0.004,Y -326.636,Z 1214.681,A 0.000,B 0.000,C 90.000,E1 122.594} C_DIS
LIN {X -0.031,Y -338.699,Z 1214.664,A 0.000,B 0.000,C 90.000,E1 119.461} C_DIS
LIN {X -0.037,Y -350.958,Z 1214.648,A 0.000,B 0.000,C 90.000,E1 116.693} C_DIS
LIN {X 0.168,Y -364.699,Z 1214.633,A 0.000,B 0.000,C 90.000,E1 113.951} C_DIS
LIN {X 0.205,Y -378.258,Z 1214.620,A 0.000,B 0.000,C 90.000,E1 111.589} C_DIS
LIN {X -0.060,Y -393.182,Z 1214.607,A 0.000,B 0.000,C 90.000,E1 109.322} C_DIS
LIN {X 0.159,Y -409.574,Z 1214.595,A 0.000,B 0.000,C 90.000,E1 107.040} C_DIS
LIN {X -0.126,Y -427.551,Z 1214.583,A 0.000,B 0.000,C 90.000,E1 104.883} C_DIS
LIN {X -0.200,Y -447.089,Z 1214.571,A 0.000,B 0.000,C 90.000,E1 102.771} C_DIS
LIN {X 0.025,Y -467.356,Z 1214.560,A 0.000,B 0.000,C 90.000,E1 100.782} C_DIS
LIN {X 0.083,Y -472.401,Z 1214.557,A 0.000,B 0.000,C 90.000,E1 100.310} C_DIS
LIN {X 0.131,Y -474.306,Z 1214.556,A 0.000,B 0.000,C 90.000,E1 100.074} C_DIS
LIN {X -0.090,Y -475.890,Z 1214.555,A 0.000,B 0.000,C 90.000,E1 99.849} C_DIS
LIN {X -0.230,Y -477.077,Z 1214.553,A 0.000,B 0.000,C 90.000,E1 99.613} C_DIS
LIN {X -0.097,Y -478.515,Z 1214.550,A 0.000,B 0.000,C 90.000,E1 99.095} C_DIS
LIN {X 0.118,Y -478.918,Z 1214.548,A 0.000,B 0.000,C 90.000,E1 98.568} C_DIS
LIN {X -0.205,Y -478.351,Z 1214.545,A 0.000,B 0.000,C 90.000,E1 98.106} C_DIS
LIN {X -0.050,Y -476.726,Z 1214.542,A 0.000,B 0.000,C 90.000,E1 97.587} C_DIS
LIN {X -0.180,Y -475.428,Z 1214.541,A 0.000,B 0.000,C 90.000,E1 97.352} C_DIS
LIN {X 0.186,Y -464.538,Z 1214.532,A 0.000,B 0.000,C 90.000,E1 95.796} C_DIS
LIN {X 0.067,Y -445.009,Z 1214.517,A 0.000,B 0.000,C 90.000,E1 92.980} C_DIS
LIN {X 0.162,Y -426.955,Z 1214.500,A 0.000,B 0.000,C 90.000,E1 90.057} C_DIS
LIN {X 0.040,Y -412.063,Z 1214.485,A 0.000,B 0.000,C 90.000,E1 87.364} C_DIS
LIN {X -0.148,Y -400.566,Z 1214.473,A 0.000,B 0.000,C 90.000,E1 85.179} C_DIS
LIN {X 0.171,Y -390.344,Z 1214.462,A 0.000,B 0.000,C 90.000,E1 83.166} C_DIS
LIN {X -0.028,Y -380.090,Z 1214.451,A 0.000,B 0.000,C 90.000,E1 81.197} C_DIS
LIN {X -0.001,Y -372.578,Z 1214.443,A 0.000,B 0.000,C 90.000,E1 79.746} C_DIS
LIN {X -0.042,Y -363.257,Z 1214.433,A 0.000,B 0.000,C 90.000,E1 77.993} C_DIS
LIN {X 0.173,Y -353.701,Z 1214.423,A 0.000,B 0.000,C 90.000,E1 76.172} C_DIS
LIN {X -0.130,Y -342.497,Z 1214.411,A 0.000,B 0.000,C 90.000,E1 74.102} C_DIS
LIN {X 0.146,Y -329.748,Z 1214.398,A 0.000,B 0.000,C 90.000,E1 71.583} C_DIS
LIN {X -0.052,Y -315.878,Z 1214.382,A 0.000,B 0.000,C 90.000,E1 68.773} C_DIS
LIN {X 0.084,Y -300.061,Z 1214.362,A 0.000,B 0.000,C 90.000,E1 65.177} C_DIS
LIN {X 0.068,Y -286.847,Z 1214.344,A 0.000,B 0.000,C 90.000,E1 61.847} C_DIS
LIN {X -0.043,Y -274.504,Z 1214.325,A 0.000,B 0.000,C 90.000,E1 58.456} C_DIS
LIN {X 0.003,Y -264.248,Z 1214.307,A 0.000,B 0.000,C 90.000,E1 55.308} C_DIS
LIN {X 0.050,Y -253.658,Z 1214.287,A 0.000,B 0.000,C 90.000,E1 51.743} C_DIS
LIN {X -0.139,Y -243.781,Z 1214.267,A 0.000,B 0.000,C 90.000,E1 48.162} C_DIS
LIN {X 0.064,Y -236.262,Z 1214.251,A 0.000,B 0.000,C 90.000,E1 45.162} C_DIS
LIN {X 0.077,Y -229.064,Z 1214.234,A 0.000,B 0.000,C 90.000,E1 42.162} C_DIS
LIN {X -0.038,Y -220.470,Z 1214.213,A 0.000,B 0.000,C 90.000,E1 38.382} C_DIS
LIN {X -0.129,Y -214.315,Z 1214.196,A 0.000,B 0.000,C 90.000,E1 35.311} C_DIS
LIN {X 0.050,Y -207.610,Z 1214.174,A 0.000,B 0.000,C 90.000,E1 31.337} C_DIS
LIN {X -0.053,Y -201.879,Z 1214.152,A 0.000,B 0.000,C 90.000,E1 27.385} C_DIS
LIN {X 0.020,Y -196.954,Z 1214.130,A 0.000,B 0.000,C 90.000,E1 23.334} C_DIS
LIN {X -0.004,Y -192.781,Z 1214.107,A 0.000,B 0.000,C 90.000,E1 19.268} C_DIS
LIN {X -0.076,Y -188.936,Z 1214.080,A 0.000,B 0.000,C 90.000,E1 14.356} C_DIS
LIN {X 0.053,Y -186.083,Z 1214.047,A 0.000,B 0.000,C 90.000,E1 8.511} C_DIS
LIN {X -0.055,Y -187.052,Z 1213.970,A 0.000,B 0.000,C 90.000,E1 354.546} C_DIS
LIN {X -0.059,Y -189.950,Z 1213.942,A 0.000,B 0.000,C 90.000,E1 349.567} C_DIS
LIN {X -0.080,Y -194.234,Z 1213.914,A 0.000,B 0.000,C 90.000,E1 344.629} C_DIS
LIN {X -0.091,Y -198.744,Z 1213.892,A 0.000,B 0.000,C 90.000,E1 340.550} C_DIS
LIN {X -0.003,Y -204.022,Z 1213.869,A 0.000,B 0.000,C 90.000,E1 336.485} C_DIS
LIN {X 0.020,Y -209.920,Z 1213.847,A 0.000,B 0.000,C 90.000,E1 332.487} C_DIS
LIN {X 0.064,Y -216.285,Z 1213.825,A 0.000,B 0.000,C 90.000,E1 328.535} C_DIS
LIN {X -0.091,Y -223.223,Z 1213.804,A 0.000,B 0.000,C 90.000,E1 324.689} C_DIS
LIN {X -0.080,Y -229.304,Z 1213.787,A 0.000,B 0.000,C 90.000,E1 321.618} C_DIS
LIN {X -0.085,Y -237.694,Z 1213.766,A 0.000,B 0.000,C 90.000,E1 317.838} C_DIS
LIN {X 0.012,Y -245.363,Z 1213.749,A 0.000,B 0.000,C 90.000,E1 314.838} C_DIS
LIN {X -0.010,Y -254.275,Z 1213.733,A 0.000,B 0.000,C 90.000,E1 311.919} C_DIS
LIN {X -0.001,Y -263.224,Z 1213.719,A 0.000,B 0.000,C 90.000,E1 309.402} C_DIS
LIN {X -0.007,Y -274.415,Z 1213.703,A 0.000,B 0.000,C 90.000,E1 306.583} C_DIS
LIN {X -0.086,Y -288.795,Z 1213.686,A 0.000,B 0.000,C 90.000,E1 303.499} C_DIS
LIN {X 0.028,Y -304.966,Z 1213.669,A 0.000,B 0.000,C 90.000,E1 300.463} C_DIS
LIN {X 0.116,Y -310.910,Z 1213.664,A 0.000,B 0.000,C 90.000,E1 299.461} C_DIS
LIN {X 0.021,Y -319.961,Z 1213.657,A 0.000,B 0.000,C 90.000,E1 298.180} C_DIS
LIN {X -0.041,Y -335.002,Z 1213.646,A 0.000,B 0.000,C 90.000,E1 296.283} C_DIS
LIN {X -0.169,Y -353.432,Z 1213.634,A 0.000,B 0.000,C 90.000,E1 294.207} C_DIS
LIN {X -0.019,Y -371.872,Z 1213.623,A 0.000,B 0.000,C 90.000,E1 292.206} C_DIS
LIN {X 0.072,Y -387.785,Z 1213.614,A 0.000,B 0.000,C 90.000,E1 290.556} C_DIS
LIN {X -0.094,Y -400.696,Z 1213.607,A 0.000,B 0.000,C 90.000,E1 289.268} C_DIS
LIN {X -0.057,Y -413.691,Z 1213.600,A 0.000,B 0.000,C 90.000,E1 287.946} C_DIS
LIN {X -0.169,Y -423.667,Z 1213.594,A 0.000,B 0.000,C 90.000,E1 286.913} C_DIS
LIN {X 0.033,Y -430.816,Z 1213.589,A 0.000,B 0.000,C 90.000,E1 286.079} C_DIS
LIN {X -0.165,Y -437.435,Z 1213.585,A 0.000,B 0.000,C 90.000,E1 285.300} C_DIS
LIN {X 0.012,Y -443.410,Z 1213.580,A 0.000,B 0.000,C 90.000,E1 284.481} C_DIS
LIN {X -0.080,Y -448.834,Z 1213.576,A 0.000,B 0.000,C 90.000,E1 283.703} C_DIS
LIN {X 0.210,Y -453.615,Z 1213.572,A 0.000,B 0.000,C 90.000,E1 282.883} C_DIS
LIN {X 0.100,Y -457.659,Z 1213.567,A 0.000,B 0.000,C 90.000,E1 282.119} C_DIS
LIN {X -0.065,Y -461.017,Z 1213.563,A 0.000,B 0.000,C 90.000,E1 281.366} C_DIS
LIN {X -0.112,Y -463.787,Z 1213.559,A 0.000,B 0.000,C 90.000,E1 280.602} C_DIS
LIN {X 0.016,Y -465.307,Z 1213.556,A 0.000,B 0.000,C 90.000,E1 280.074} C_DIS
LIN {X 0.073,Y -466.566,Z 1213.553,A 0.000,B 0.000,C 90.000,E1 279.557} C_DIS
LIN {X 0.217,Y -467.505,Z 1213.550,A 0.000,B 0.000,C 90.000,E1 279.029} C_DIS
LIN {X -0.167,Y -468.199,Z 1213.547,A 0.000,B 0.000,C 90.000,E1 278.568} C_DIS
LIN {X -0.082,Y -468.644,Z 1213.545,A 0.000,B 0.000,C 90.000,E1 278.049} C_DIS
LIN {X 0.009,Y -468.807,Z 1213.542,A 0.000,B 0.000,C 90.000,E1 277.530} C_DIS
LIN {X 0.105,Y -468.630,Z 1213.539,A 0.000,B 0.000,C 90.000,E1 277.011} C_DIS
LIN {X 0.256,Y -468.054,Z 1213.536,A 0.000,B 0.000,C 90.000,E1 276.486} C_DIS
LIN {X -0.118,Y -467.073,Z 1213.533,A 0.000,B 0.000,C 90.000,E1 276.024} C_DIS
LIN {X -0.074,Y -465.690,Z 1213.531,A 0.000,B 0.000,C 90.000,E1 275.511} C_DIS
LIN {X 0.012,Y -463.863,Z 1213.528,A 0.000,B 0.000,C 90.000,E1 274.992} C_DIS
LIN {X 0.086,Y -461.482,Z 1213.525,A 0.000,B 0.000,C 90.000,E1 274.473} C_DIS
LIN {X 0.141,Y -458.485,Z 1213.522,A 0.000,B 0.000,C 90.000,E1 273.955} C_DIS
LIN {X 0.148,Y -454.694,Z 1213.519,A 0.000,B 0.000,C 90.000,E1 273.440} C_DIS
LIN {X 0.164,Y -449.793,Z 1213.516,A 0.000,B 0.000,C 90.000,E1 272.922} C_DIS
LIN {X -0.011,Y -447.013,Z 1213.515,A 0.000,B 0.000,C 90.000,E1 272.694} C_DIS
LIN {X -0.063,Y -440.770,Z 1213.512,A 0.000,B 0.000,C 90.000,E1 272.236} C_DIS
LIN {X 0.012,Y -433.971,Z 1213.510,A 0.000,B 0.000,C 90.000,E1 271.835} C_DIS
LIN {X 0.212,Y -426.698,Z 1213.508,A 0.000,B 0.000,C 90.000,E1 271.489} C_DIS
LIN {X -0.013,Y -419.727,Z 1213.507,A 0.000,B 0.000,C 90.000,E1 271.260} C_DIS
LIN {X 0.121,Y -409.398,Z 1213.505,A 0.000,B 0.000,C 90.000,E1 270.917} C_DIS
LIN {X -0.170,Y -399.095,Z 1213.504,A 0.000,B 0.000,C 90.000,E1 270.688} C_DIS
LIN {X -0.040,Y -391.810,Z 1213.503,A 0.000,B 0.000,C 90.000,E1 270.516} C_DIS
LIN {X -0.122,Y -383.168,Z 1213.502,A 0.000,B 0.000,C 90.000,E1 270.401} C_DIS
LIN {X -0.023,Y -373.221,Z 1213.502,A 0.000,B 0.000,C 90.000,E1 270.286} C_DIS
LIN {X 0.134,Y -365.946,Z 1213.501,A 0.000,B 0.000,C 90.000,E1 270.229} C_DIS
LIN {X 0.032,Y -181.581,Z 1213.501,A 0.000,B 0.000,C 90.000,E1 270.229} C_DIS
LIN {X 0.010,Y -180.818,Z 1213.471,A 0.000,B 0.000,C 90.000,E1 264.837} C_DIS
LIN {X 0.086,Y -178.921,Z 1213.443,A 0.000,B 0.000,C 90.000,E1 259.746} C_DIS
LIN {X -0.004,Y -175.967,Z 1213.415,A 0.000,B 0.000,C 90.000,E1 254.685} C_DIS
LIN {X -0.057,Y -175.448,Z 1213.410,A 0.000,B 0.000,C 90.000,E1 253.850} C_DIS
LIN {X -0.048,Y -172.202,Z 1213.386,A 0.000,B 0.000,C 90.000,E1 249.571} C_DIS
LIN {X -0.070,Y -171.676,Z 1213.382,A 0.000,B 0.000,C 90.000,E1 248.720} C_DIS
LIN {X -0.079,Y -167.902,Z 1213.358,A 0.000,B 0.000,C 90.000,E1 244.409} C_DIS
LIN {X -0.060,Y -166.642,Z 1213.348,A 0.000,B 0.000,C 90.000,E1 242.666} C_DIS
LIN {X -0.005,Y -162.626,Z 1213.324,A 0.000,B 0.000,C 90.000,E1 238.280} C_DIS
LIN {X 0.054,Y -161.314,Z 1213.314,A 0.000,B 0.000,C 90.000,E1 236.501} C_DIS
LIN {X -0.037,Y -157.310,Z 1213.289,A 0.000,B 0.000,C 90.000,E1 232.110} C_DIS
LIN {X -0.103,Y -155.288,Z 1213.275,A 0.000,B 0.000,C 90.000,E1 229.461} C_DIS
LIN {X 0.043,Y -151.650,Z 1213.250,A 0.000,B 0.000,C 90.000,E1 224.919} C_DIS
LIN {X -0.020,Y -150.519,Z 1213.240,A 0.000,B 0.000,C 90.000,E1 223.137} C_DIS
LIN {X 0.004,Y -147.243,Z 1213.214,A 0.000,B 0.000,C 90.000,E1 218.588} C_DIS
LIN {X -0.032,Y -145.267,Z 1213.194,A 0.000,B 0.000,C 90.000,E1 214.945} C_DIS
LIN {X 0.003,Y -142.376,Z 1213.163,A 0.000,B 0.000,C 90.000,E1 209.411} C_DIS
LIN {X 0.052,Y -141.352,Z 1213.148,A 0.000,B 0.000,C 90.000,E1 206.616} C_DIS
LIN {X 0.036,Y -139.340,Z 1213.112,A 0.000,B 0.000,C 90.000,E1 200.120} C_DIS
LIN {X -0.046,Y -139.006,Z 1213.102,A 0.000,B 0.000,C 90.000,E1 198.290} C_DIS
LIN {X 0.042,Y -138.340,Z 1213.055,A 0.000,B 0.000,C 90.000,E1 189.849} C_DIS
LIN {X 0.064,Y -139.404,Z 1213.008,A 0.000,B 0.000,C 90.000,E1 181.432} C_DIS
LIN {X -0.022,Y -141.310,Z 1212.972,A 0.000,B 0.000,C 90.000,E1 174.951} C_DIS
LIN {X -0.065,Y -142.671,Z 1212.956,A 0.000,B 0.000,C 90.000,E1 172.186} C_DIS
LIN {X 0.057,Y -145.021,Z 1212.931,A 0.000,B 0.000,C 90.000,E1 167.521} C_DIS
LIN {X 0.014,Y -147.647,Z 1212.910,A 0.000,B 0.000,C 90.000,E1 163.866} C_DIS
LIN {X -0.051,Y -150.282,Z 1212.890,A 0.000,B 0.000,C 90.000,E1 160.242} C_DIS
LIN {X -0.038,Y -153.687,Z 1212.870,A 0.000,B 0.000,C 90.000,E1 156.613} C_DIS
LIN {X 0.018,Y -157.102,Z 1212.850,A 0.000,B 0.000,C 90.000,E1 152.999} C_DIS
LIN {X -0.044,Y -161.241,Z 1212.830,A 0.000,B 0.000,C 90.000,E1 149.459} C_DIS
LIN {X 0.041,Y -163.328,Z 1212.820,A 0.000,B 0.000,C 90.000,E1 147.661} C_DIS
LIN {X -0.088,Y -167.781,Z 1212.801,A 0.000,B 0.000,C 90.000,E1 144.196} C_DIS
LIN {X 0.064,Y -171.596,Z 1212.786,A 0.000,B 0.000,C 90.000,E1 141.537} C_DIS
LIN {X -0.006,Y -176.548,Z 1212.767,A 0.000,B 0.000,C 90.000,E1 138.119} C_DIS
LIN {X -0.014,Y -180.846,Z 1212.753,A 0.000,B 0.000,C 90.000,E1 135.567} C_DIS
LIN {X -0.030,Y -186.257,Z 1212.734,A 0.000,B 0.000,C 90.000,E1 132.204} C_DIS
LIN {X -0.092,Y -190.894,Z 1212.721,A 0.000,B 0.000,C 90.000,E1 129.725} C_DIS
LIN {X -0.059,Y -196.658,Z 1212.702,A 0.000,B 0.000,C 90.000,E1 126.423} C_DIS
LIN {X -0.031,Y -201.171,Z 1212.689,A 0.000,B 0.000,C 90.000,E1 124.119} C_DIS
LIN {X -0.048,Y -201.315,Z 1212.689,A 0.000,B 0.000,C 90.000,E1 124.040} C_DIS
LIN {X 0.148,Y -311.501,Z 1212.689,A 0.000,B 0.000,C 90.000,E1 123.992} C_DIS
LIN {X -0.146,Y -314.108,Z 1212.689,A 0.000,B 0.000,C 90.000,E1 123.992} C_DIS
LIN {X 0.100,Y -317.440,Z 1212.688,A 0.000,B 0.000,C 90.000,E1 123.785} C_DIS
LIN {X 0.019,Y -320.953,Z 1212.686,A 0.000,B 0.000,C 90.000,E1 123.499} C_DIS
LIN {X 0.010,Y -324.553,Z 1212.683,A 0.000,B 0.000,C 90.000,E1 123.007} C_DIS
LIN {X 0.095,Y -326.184,Z 1212.682,A 0.000,B 0.000,C 90.000,E1 122.673} C_DIS
LIN {X 0.000,Y -333.314,Z 1212.671,A 0.000,B 0.000,C 90.000,E1 120.797} C_DIS
LIN {X -0.138,Y -344.903,Z 1212.656,A 0.000,B 0.000,C 90.000,E1 118.025} C_DIS
LIN {X -0.120,Y -357.919,Z 1212.640,A 0.000,B 0.000,C 90.000,E1 115.283} C_DIS
LIN {X -0.113,Y -370.785,Z 1212.627,A 0.000,B 0.000,C 90.000,E1 112.898} C_DIS
LIN {X -0.067,Y -384.964,Z 1212.614,A 0.000,B 0.000,C 90.000,E1 110.556} C_DIS
LIN {X 0.202,Y -400.553,Z 1212.601,A 0.000,B 0.000,C 90.000,E1 108.236} C_DIS
LIN {X 0.106,Y -417.663,Z 1212.589,A 0.000,B 0.000,C 90.000,E1 106.024} C_DIS
LIN {X -0.102,Y -436.416,Z 1212.577,A 0.000,B 0.000,C 90.000,E1 103.883} C_DIS
LIN {X -0.076,Y -456.370,Z 1212.566,A 0.000,B 0.000,C 90.000,E1 101.827} C_DIS
LIN {X 0.182,Y -471.684,Z 1212.558,A 0.000,B 0.000,C 90.000,E1 100.366} C_DIS
LIN {X 0.140,Y -473.743,Z 1212.556,A 0.000,B 0.000,C 90.000,E1 100.141} C_DIS
LIN {X 0.002,Y -475.440,Z 1212.555,A 0.000,B 0.000,C 90.000,E1 99.905} C_DIS
LIN {X -0.140,Y -476.713,Z 1212.554,A 0.000,B 0.000,C 90.000,E1 99.670} C_DIS
LIN {X -0.012,Y -478.287,Z 1212.551,A 0.000,B 0.000,C 90.000,E1 99.151} C_DIS
LIN {X 0.202,Y -478.805,Z 1212.548,A 0.000,B 0.000,C 90.000,E1 98.624} C_DIS
LIN {X -0.123,Y -478.354,Z 1212.545,A 0.000,B 0.000,C 90.000,E1 98.163} C_DIS
LIN {X 0.030,Y -476.864,Z 1212.542,A 0.000,B 0.000,C 90.000,E1 97.644} C_DIS
LIN {X -0.100,Y -475.654,Z 1212.541,A 0.000,B 0.000,C 90.000,E1 97.409} C_DIS
LIN {X 0.181,Y -474.041,Z 1212.540,A 0.000,B 0.000,C 90.000,E1 97.125} C_DIS
LIN {X -0.095,Y -457.632,Z 1212.527,A 0.000,B 0.000,C 90.000,E1 94.878} C_DIS
LIN {X -0.171,Y -440.231,Z 1212.513,A 0.000,B 0.000,C 90.000,E1 92.293} C_DIS
LIN {X 0.092,Y -424.161,Z 1212.498,A 0.000,B 0.000,C 90.000,E1 89.599} C_DIS
LIN {X -0.188,Y -410.853,Z 1212.484,A 0.000,B 0.000,C 90.000,E1 87.192} C_DIS
LIN {X -0.003,Y -399.343,Z 1212.472,A 0.000,B 0.000,C 90.000,E1 84.951} C_DIS
LIN {X -0.109,Y -389.112,Z 1212.461,A 0.000,B 0.000,C 90.000,E1 82.996} C_DIS
LIN {X 0.047,Y -378.853,Z 1212.450,A 0.000,B 0.000,C 90.000,E1 80.971} C_DIS
LIN {X 0.111,Y -371.292,Z 1212.442,A 0.000,B 0.000,C 90.000,E1 79.511} C_DIS
LIN {X 0.046,Y -361.939,Z 1212.432,A 0.000,B 0.000,C 90.000,E1 77.757} C_DIS
LIN {X -0.160,Y -350.781,Z 1212.420,A 0.000,B 0.000,C 90.000,E1 75.700} C_DIS
LIN {X -0.093,Y -339.575,Z 1212.409,A 0.000,B 0.000,C 90.000,E1 73.559} C_DIS
LIN {X 0.110,Y -326.853,Z 1212.395,A 0.000,B 0.000,C 90.000,E1 71.040} C_DIS
LIN {X -0.048,Y -313.154,Z 1212.379,A 0.000,B 0.000,C 90.000,E1 68.209} C_DIS
LIN {X 0.126,Y -297.552,Z 1212.359,A 0.000,B 0.000,C 90.000,E1 64.588} C_DIS
LIN {X 0.067,Y -285.776,Z 1212.342,A 0.000,B 0.000,C 90.000,E1 61.591} C_DIS
LIN {X -0.081,Y -273.484,Z 1212.323,A 0.000,B 0.000,C 90.000,E1 58.201} C_DIS
LIN {X -0.073,Y -263.254,Z 1212.306,A 0.000,B 0.000,C 90.000,E1 55.055} C_DIS
LIN {X 0.064,Y -253.730,Z 1212.288,A 0.000,B 0.000,C 90.000,E1 51.823} C_DIS
LIN {X -0.126,Y -243.789,Z 1212.268,A 0.000,B 0.000,C 90.000,E1 48.243} C_DIS
LIN {X 0.076,Y -236.218,Z 1212.251,A 0.000,B 0.000,C 90.000,E1 45.243} C_DIS
LIN {X -0.082,Y -228.956,Z 1212.235,A 0.000,B 0.000,C 90.000,E1 42.285} C_DIS
LIN {X -0.030,Y -220.341,Z 1212.214,A 0.000,B 0.000,C 90.000,E1 38.463} C_DIS
LIN {X 0.003,Y -214.183,Z 1212.196,A 0.000,B 0.000,C 90.000,E1 35.358} C_DIS
LIN {X 0.058,Y -207.484,Z 1212.175,A 0.000,B 0.000,C 90.000,E1 31.416} C_DIS
LIN {X -0.044,Y -201.754,Z 1212.152,A 0.000,B 0.000,C 90.000,E1 27.462} C_DIS
LIN {X 0.110,Y -196.781,Z 1212.130,A 0.000,B 0.000,C 90.000,E1 23.387} C_DIS
LIN {X 0.074,Y -192.578,Z 1212.107,A 0.000,B 0.000,C 90.000,E1 19.322} C_DIS
LIN {X -0.012,Y -188.685,Z 1212.080,A 0.000,B 0.000,C 90.000,E1 14.411} C_DIS
LIN {X -0.084,Y -185.781,Z 1212.048,A 0.000,B 0.000,C 90.000,E1 8.624} C_DIS
LIN {X -0.067,Y -186.719,Z 1211.970,A 0.000,B 0.000,C 90.000,E1 354.546} C_DIS
LIN {X 0.103,Y -189.629,Z 1211.942,A 0.000,B 0.000,C 90.000,E1 349.511} C_DIS
LIN {X 0.027,Y -193.126,Z 1211.919,A 0.000,B 0.000,C 90.000,E1 345.408} C_DIS
LIN {X -0.018,Y -197.487,Z 1211.896,A 0.000,B 0.000,C 90.000,E1 341.329} C_DIS
LIN {X -0.035,Y -202.641,Z 1211.874,A 0.000,B 0.000,C 90.000,E1 337.283} C_DIS
LIN {X 0.047,Y -208.436,Z 1211.851,A 0.000,B 0.000,C 90.000,E1 333.256} C_DIS
LIN {X -0.095,Y -213.455,Z 1211.834,A 0.000,B 0.000,C 90.000,E1 330.127} C_DIS
LIN {X -0.089,Y -220.118,Z 1211.812,A 0.000,B 0.000,C 90.000,E1 326.215} C_DIS
LIN {X -0.056,Y -227.536,Z 1211.791,A 0.000,B 0.000,C 90.000,E1 322.351} C_DIS
LIN {X 0.060,Y -235.708,Z 1211.770,A 0.000,B 0.000,C 90.000,E1 318.528} C_DIS
LIN {X 0.093,Y -244.180,Z 1211.751,A 0.000,B 0.000,C 90.000,E1 315.162} C_DIS
LIN {X 0.042,Y -253.019,Z 1211.735,A 0.000,B 0.000,C 90.000,E1 312.243} C_DIS
LIN {X 0.075,Y -263.205,Z 1211.719,A 0.000,B 0.000,C 90.000,E1 309.358} C_DIS
LIN {X -0.141,Y -274.433,Z 1211.703,A 0.000,B 0.000,C 90.000,E1 306.583} C_DIS
LIN {X 0.014,Y -288.818,Z 1211.686,A 0.000,B 0.000,C 90.000,E1 303.452} C_DIS
LIN {X -0.120,Y -305.012,Z 1211.669,A 0.000,B 0.000,C 90.000,E1 300.463} C_DIS
LIN {X -0.034,Y -311.013,Z 1211.664,A 0.000,B 0.000,C 90.000,E1 299.461} C_DIS
LIN {X 0.019,Y -319.997,Z 1211.656,A 0.000,B 0.000,C 90.000,E1 298.153} C_DIS
LIN {X 0.099,Y -335.007,Z 1211.646,A 0.000,B 0.000,C 90.000,E1 296.232} C_DIS
LIN {X -0.176,Y -350.924,Z 1211.636,A 0.000,B 0.000,C 90.000,E1 294.463} C_DIS
LIN {X 0.023,Y -369.164,Z 1211.625,A 0.000,B 0.000,C 90.000,E1 292.461} C_DIS
LIN {X 0.063,Y -387.660,Z 1211.614,A 0.000,B 0.000,C 90.000,E1 290.556} C_DIS
LIN {X -0.068,Y -400.585,Z 1211.607,A 0.000,B 0.000,C 90.000,E1 289.268} C_DIS
LIN {X -0.020,Y -413.599,Z 1211.600,A 0.000,B 0.000,C 90.000,E1 287.946} C_DIS
LIN {X -0.134,Y -423.589,Z 1211.594,A 0.000,B 0.000,C 90.000,E1 286.913} C_DIS
LIN {X 0.061,Y -430.779,Z 1211.589,A 0.000,B 0.000,C 90.000,E1 286.079} C_DIS
LIN {X -0.137,Y -437.397,Z 1211.585,A 0.000,B 0.000,C 90.000,E1 285.300} C_DIS
LIN {X 0.040,Y -443.381,Z 1211.580,A 0.000,B 0.000,C 90.000,E1 284.481} C_DIS
LIN {X -0.052,Y -448.815,Z 1211.576,A 0.000,B 0.000,C 90.000,E1 283.703} C_DIS
LIN {X 0.239,Y -453.610,Z 1211.572,A 0.000,B 0.000,C 90.000,E1 282.883} C_DIS
LIN {X 0.129,Y -457.659,Z 1211.567,A 0.000,B 0.000,C 90.000,E1 282.119} C_DIS
LIN {X -0.036,Y -461.021,Z 1211.563,A 0.000,B 0.000,C 90.000,E1 281.366} C_DIS
LIN {X -0.083,Y -463.819,Z 1211.559,A 0.000,B 0.000,C 90.000,E1 280.602} C_DIS
LIN {X 0.045,Y -465.321,Z 1211.556,A 0.000,B 0.000,C 90.000,E1 280.074} C_DIS
LIN {X 0.103,Y -466.577,Z 1211.553,A 0.000,B 0.000,C 90.000,E1 279.557} C_DIS
LIN {X 0.247,Y -467.527,Z 1211.550,A 0.000,B 0.000,C 90.000,E1 279.029} C_DIS
LIN {X -0.137,Y -468.222,Z 1211.547,A 0.000,B 0.000,C 90.000,E1 278.568} C_DIS
LIN {X -0.052,Y -468.700,Z 1211.545,A 0.000,B 0.000,C 90.000,E1 278.049} C_DIS
LIN {X 0.040,Y -468.881,Z 1211.542,A 0.000,B 0.000,C 90.000,E1 277.530} C_DIS
LIN {X 0.136,Y -468.714,Z 1211.539,A 0.000,B 0.000,C 90.000,E1 277.011} C_DIS
LIN {X -0.179,Y -468.186,Z 1211.536,A 0.000,B 0.000,C 90.000,E1 276.543} C_DIS
LIN {X -0.135,Y -467.230,Z 1211.533,A 0.000,B 0.000,C 90.000,E1 276.030} C_DIS
LIN {X -0.041,Y -465.878,Z 1211.531,A 0.000,B 0.000,C 90.000,E1 275.511} C_DIS
LIN {X 0.044,Y -464.088,Z 1211.528,A 0.000,B 0.000,C 90.000,E1 274.992} C_DIS
LIN {X 0.120,Y -461.748,Z 1211.525,A 0.000,B 0.000,C 90.000,E1 274.473} C_DIS
LIN {X 0.175,Y -458.770,Z 1211.522,A 0.000,B 0.000,C 90.000,E1 273.955} C_DIS
LIN {X 0.185,Y -455.028,Z 1211.519,A 0.000,B 0.000,C 90.000,E1 273.440} C_DIS
LIN {X -0.044,Y -452.788,Z 1211.518,A 0.000,B 0.000,C 90.000,E1 273.212} C_DIS
LIN {X 0.026,Y -447.419,Z 1211.515,A 0.000,B 0.000,C 90.000,E1 272.694} C_DIS
LIN {X -0.039,Y -441.221,Z 1211.512,A 0.000,B 0.000,C 90.000,E1 272.236} C_DIS
LIN {X 0.070,Y -437.787,Z 1211.511,A 0.000,B 0.000,C 90.000,E1 272.007} C_DIS
LIN {X -0.048,Y -430.548,Z 1211.509,A 0.000,B 0.000,C 90.000,E1 271.661} C_DIS
LIN {X -0.008,Y -423.433,Z 1211.508,A 0.000,B 0.000,C 90.000,E1 271.375} C_DIS
LIN {X 0.023,Y -413.201,Z 1211.506,A 0.000,B 0.000,C 90.000,E1 271.031} C_DIS
LIN {X -0.018,Y -402.825,Z 1211.504,A 0.000,B 0.000,C 90.000,E1 270.745} C_DIS
LIN {X -0.057,Y -392.431,Z 1211.503,A 0.000,B 0.000,C 90.000,E1 270.516} C_DIS
LIN {X -0.099,Y -379.900,Z 1211.502,A 0.000,B 0.000,C 90.000,E1 270.344} C_DIS
LIN {X -0.172,Y -371.684,Z 1211.501,A 0.000,B 0.000,C 90.000,E1 270.286} C_DIS
LIN {X 0.002,Y -364.351,Z 1211.501,A 0.000,B 0.000,C 90.000,E1 270.229} C_DIS
LIN {X -0.022,Y -181.580,Z 1211.501,A 0.000,B 0.000,C 90.000,E1 270.229} C_DIS
LIN {X 0.007,Y -180.886,Z 1211.473,A 0.000,B 0.000,C 90.000,E1 265.122} C_DIS
LIN {X 0.066,Y -179.007,Z 1211.445,A 0.000,B 0.000,C 90.000,E1 260.038} C_DIS
LIN {X -0.016,Y -178.616,Z 1211.440,A 0.000,B 0.000,C 90.000,E1 259.218} C_DIS
LIN {X 0.053,Y -175.668,Z 1211.412,A 0.000,B 0.000,C 90.000,E1 254.102} C_DIS
LIN {X 0.057,Y -172.385,Z 1211.388,A 0.000,B 0.000,C 90.000,E1 249.826} C_DIS
LIN {X 0.071,Y -171.186,Z 1211.379,A 0.000,B 0.000,C 90.000,E1 248.103} C_DIS
LIN {X -0.036,Y -167.478,Z 1211.354,A 0.000,B 0.000,C 90.000,E1 243.819} C_DIS
LIN {X -0.029,Y -166.875,Z 1211.350,A 0.000,B 0.000,C 90.000,E1 242.948} C_DIS
LIN {X -0.037,Y -162.179,Z 1211.321,A 0.000,B 0.000,C 90.000,E1 237.709} C_DIS
LIN {X 0.021,Y -160.745,Z 1211.311,A 0.000,B 0.000,C 90.000,E1 235.928} C_DIS
LIN {X 0.000,Y -157.545,Z 1211.291,A 0.000,B 0.000,C 90.000,E1 232.396} C_DIS
LIN {X -0.062,Y -155.573,Z 1211.276,A 0.000,B 0.000,C 90.000,E1 229.747} C_DIS
LIN {X -0.009,Y -151.860,Z 1211.251,A 0.000,B 0.000,C 90.000,E1 225.243} C_DIS
LIN {X 0.004,Y -150.081,Z 1211.236,A 0.000,B 0.000,C 90.000,E1 222.528} C_DIS
LIN {X 0.038,Y -146.885,Z 1211.211,A 0.000,B 0.000,C 90.000,E1 217.971} C_DIS
LIN {X 0.026,Y -145.471,Z 1211.196,A 0.000,B 0.000,C 90.000,E1 215.231} C_DIS
LIN {X -0.056,Y -142.883,Z 1211.170,A 0.000,B 0.000,C 90.000,E1 210.669} C_DIS
LIN {X 0.001,Y -141.502,Z 1211.150,A 0.000,B 0.000,C 90.000,E1 206.950} C_DIS
LIN {X 0.050,Y -139.389,Z 1211.114,A 0.000,B 0.000,C 90.000,E1 200.429} C_DIS
LIN {X -0.031,Y -139.095,Z 1211.103,A 0.000,B 0.000,C 90.000,E1 198.598} C_DIS
LIN {X -0.038,Y -138.354,Z 1211.057,A 0.000,B 0.000,C 90.000,E1 190.197} C_DIS
LIN {X -0.046,Y -139.517,Z 1211.005,A 0.000,B 0.000,C 90.000,E1 180.859} C_DIS
LIN {X 0.035,Y -141.172,Z 1210.974,A 0.000,B 0.000,C 90.000,E1 175.241} C_DIS
LIN {X 0.006,Y -142.551,Z 1210.958,A 0.000,B 0.000,C 90.000,E1 172.470} C_DIS
LIN {X -0.069,Y -144.827,Z 1210.932,A 0.000,B 0.000,C 90.000,E1 167.881} C_DIS
LIN {X 0.061,Y -147.450,Z 1210.912,A 0.000,B 0.000,C 90.000,E1 164.157} C_DIS
LIN {X -0.054,Y -150.032,Z 1210.892,A 0.000,B 0.000,C 90.000,E1 160.550} C_DIS
LIN {X -0.048,Y -153.369,Z 1210.872,A 0.000,B 0.000,C 90.000,E1 156.922} C_DIS
LIN {X 0.001,Y -155.902,Z 1210.857,A 0.000,B 0.000,C 90.000,E1 154.204} C_DIS
LIN {X -0.023,Y -159.762,Z 1210.837,A 0.000,B 0.000,C 90.000,E1 150.639} C_DIS
LIN {X -0.036,Y -162.003,Z 1210.827,A 0.000,B 0.000,C 90.000,E1 148.869} C_DIS
LIN {X 0.077,Y -166.196,Z 1210.807,A 0.000,B 0.000,C 90.000,E1 145.308} C_DIS
LIN {X 0.080,Y -171.211,Z 1210.788,A 0.000,B 0.000,C 90.000,E1 141.823} C_DIS
LIN {X 0.005,Y -176.095,Z 1210.769,A 0.000,B 0.000,C 90.000,E1 138.405} C_DIS
LIN {X -0.004,Y -180.357,Z 1210.755,A 0.000,B 0.000,C 90.000,E1 135.850} C_DIS
LIN {X 0.099,Y -185.766,Z 1210.736,A 0.000,B 0.000,C 90.000,E1 132.447} C_DIS
LIN {X 0.033,Y -190.379,Z 1210.722,A 0.000,B 0.000,C 90.000,E1 129.967} C_DIS
LIN {X -0.067,Y -197.704,Z 1210.699,A 0.000,B 0.000,C 90.000,E1 125.884} C_DIS
LIN {X 0.006,Y -201.369,Z 1210.689,A 0.000,B 0.000,C 90.000,E1 123.992} C_DIS
LIN {X -0.039,Y -311.814,Z 1210.689,A 0.000,B 0.000,C 90.000,E1 123.992} C_DIS
LIN {X 0.072,Y -316.235,Z 1210.688,A 0.000,B 0.000,C 90.000,E1 123.833} C_DIS
LIN {X 0.008,Y -318.418,Z 1210.687,A 0.000,B 0.000,C 90.000,E1 123.706} C_DIS
LIN {X 0.055,Y -321.399,Z 1210.686,A 0.000,B 0.000,C 90.000,E1 123.420} C_DIS
LIN {X 0.123,Y -325.062,Z 1210.683,A 0.000,B 0.000,C 90.000,E1 122.880} C_DIS
LIN {X -0.065,Y -326.604,Z 1210.681,A 0.000,B 0.000,C 90.000,E1 122.594} C_DIS
LIN {X -0.130,Y -339.999,Z 1210.662,A 0.000,B 0.000,C 90.000,E1 119.155} C_DIS
LIN {X 0.070,Y -352.420,Z 1210.646,A 0.000,B 0.000,C 90.000,E1 116.360} C_DIS
LIN {X 0.159,Y -366.344,Z 1210.631,A 0.000,B 0.000,C 90.000,E1 113.643} C_DIS
LIN {X -0.115,Y -380.075,Z 1210.618,A 0.000,B 0.000,C 90.000,E1 111.334} C_DIS
LIN {X -0.111,Y -395.183,Z 1210.606,A 0.000,B 0.000,C 90.000,E1 109.033} C_DIS
LIN {X -0.226,Y -411.775,Z 1210.593,A 0.000,B 0.000,C 90.000,E1 106.804} C_DIS
LIN {X -0.059,Y -429.967,Z 1210.581,A 0.000,B 0.000,C 90.000,E1 104.592} C_DIS
LIN {X -0.002,Y -449.657,Z 1210.569,A 0.000,B 0.000,C 90.000,E1 102.479} C_DIS
LIN {X -0.002,Y -472.410,Z 1210.557,A 0.000,B 0.000,C 90.000,E1 100.310} C_DIS
LIN {X 0.046,Y -474.257,Z 1210.556,A 0.000,B 0.000,C 90.000,E1 100.074} C_DIS
LIN {X -0.175,Y -475.796,Z 1210.555,A 0.000,B 0.000,C 90.000,E1 99.849} C_DIS
LIN {X 0.155,Y -476.948,Z 1210.553,A 0.000,B 0.000,C 90.000,E1 99.557} C_DIS
LIN {X -0.183,Y -478.332,Z 1210.550,A 0.000,B 0.000,C 90.000,E1 99.095} C_DIS
LIN {X 0.032,Y -478.686,Z 1210.548,A 0.000,B 0.000,C 90.000,E1 98.568} C_DIS
LIN {X 0.181,Y -478.072,Z 1210.545,A 0.000,B 0.000,C 90.000,E1 98.049} C_DIS
LIN {X -0.138,Y -476.390,Z 1210.542,A 0.000,B 0.000,C 90.000,E1 97.587} C_DIS
LIN {X 0.202,Y -475.056,Z 1210.541,A 0.000,B 0.000,C 90.000,E1 97.296} C_DIS
LIN {X 0.167,Y -460.517,Z 1210.529,A 0.000,B 0.000,C 90.000,E1 95.277} C_DIS
LIN {X -0.100,Y -441.237,Z 1210.514,A 0.000,B 0.000,C 90.000,E1 92.465} C_DIS
LIN {X 0.188,Y -425.077,Z 1210.499,A 0.000,B 0.000,C 90.000,E1 89.771} C_DIS
LIN {X -0.076,Y -411.729,Z 1210.485,A 0.000,B 0.000,C 90.000,E1 87.364} C_DIS
LIN {X 0.130,Y -400.188,Z 1210.473,A 0.000,B 0.000,C 90.000,E1 85.122} C_DIS
LIN {X 0.046,Y -389.962,Z 1210.462,A 0.000,B 0.000,C 90.000,E1 83.166} C_DIS
LIN {X -0.157,Y -379.706,Z 1210.451,A 0.000,B 0.000,C 90.000,E1 81.197} C_DIS
LIN {X -0.133,Y -372.208,Z 1210.443,A 0.000,B 0.000,C 90.000,E1 79.746} C_DIS
LIN {X 0.177,Y -362.873,Z 1210.433,A 0.000,B 0.000,C 90.000,E1 77.937} C_DIS
LIN {X -0.022,Y -351.726,Z 1210.422,A 0.000,B 0.000,C 90.000,E1 75.880} C_DIS
LIN {X 0.063,Y -340.524,Z 1210.410,A 0.000,B 0.000,C 90.000,E1 73.740} C_DIS
LIN {X -0.027,Y -327.785,Z 1210.396,A 0.000,B 0.000,C 90.000,E1 71.275} C_DIS
LIN {X 0.023,Y -314.039,Z 1210.380,A 0.000,B 0.000,C 90.000,E1 68.411} C_DIS
LIN {X -0.055,Y -298.345,Z 1210.360,A 0.000,B 0.000,C 90.000,E1 64.845} C_DIS
LIN {X -0.089,Y -286.513,Z 1210.344,A 0.000,B 0.000,C 90.000,E1 61.847} C_DIS
LIN {X 0.029,Y -274.140,Z 1210.324,A 0.000,B 0.000,C 90.000,E1 58.408} C_DIS
LIN {X 0.054,Y -263.841,Z 1210.307,A 0.000,B 0.000,C 90.000,E1 55.261} C_DIS
LIN {X 0.078,Y -253.211,Z 1210.287,A 0.000,B 0.000,C 90.000,E1 51.698} C_DIS
LIN {X 0.025,Y -243.225,Z 1210.267,A 0.000,B 0.000,C 90.000,E1 48.081} C_DIS
LIN {X -0.124,Y -235.643,Z 1210.251,A 0.000,B 0.000,C 90.000,E1 45.162} C_DIS
LIN {X -0.065,Y -226.586,Z 1210.230,A 0.000,B 0.000,C 90.000,E1 41.391} C_DIS
LIN {X 0.088,Y -218.137,Z 1210.209,A 0.000,B 0.000,C 90.000,E1 37.523} C_DIS
LIN {X 0.112,Y -212.289,Z 1210.191,A 0.000,B 0.000,C 90.000,E1 34.405} C_DIS
LIN {X 0.109,Y -205.818,Z 1210.169,A 0.000,B 0.000,C 90.000,E1 30.463} C_DIS
LIN {X 0.030,Y -200.265,Z 1210.147,A 0.000,B 0.000,C 90.000,E1 26.488} C_DIS
LIN {X -0.029,Y -195.441,Z 1210.125,A 0.000,B 0.000,C 90.000,E1 22.461} C_DIS
LIN {X 0.014,Y -191.443,Z 1210.102,A 0.000,B 0.000,C 90.000,E1 18.362} C_DIS
LIN {X 0.021,Y -187.767,Z 1210.075,A 0.000,B 0.000,C 90.000,E1 13.411} C_DIS
LIN {X 0.032,Y -185.127,Z 1210.042,A 0.000,B 0.000,C 90.000,E1 7.587} C_DIS
LIN {X -0.079,Y -186.377,Z 1209.970,A 0.000,B 0.000,C 90.000,E1 354.546} C_DIS
LIN {X 0.078,Y -189.302,Z 1209.942,A 0.000,B 0.000,C 90.000,E1 349.511} C_DIS
LIN {X -0.009,Y -192.811,Z 1209.919,A 0.000,B 0.000,C 90.000,E1 345.408} C_DIS
LIN {X -0.064,Y -197.192,Z 1209.896,A 0.000,B 0.000,C 90.000,E1 341.329} C_DIS
LIN {X 0.094,Y -202.341,Z 1209.874,A 0.000,B 0.000,C 90.000,E1 337.230} C_DIS
LIN {X -0.020,Y -208.179,Z 1209.851,A 0.000,B 0.000,C 90.000,E1 333.256} C_DIS
LIN {X 0.016,Y -213.199,Z 1209.834,A 0.000,B 0.000,C 90.000,E1 330.078} C_DIS
LIN {X 0.009,Y -219.877,Z 1209.812,A 0.000,B 0.000,C 90.000,E1 326.167} C_DIS
LIN {X -0.013,Y -227.287,Z 1209.791,A 0.000,B 0.000,C 90.000,E1 322.316} C_DIS
LIN {X -0.048,Y -235.511,Z 1209.770,A 0.000,B 0.000,C 90.000,E1 318.528} C_DIS
LIN {X -0.024,Y -244.041,Z 1209.751,A 0.000,B 0.000,C 90.000,E1 315.162} C_DIS
LIN {X -0.094,Y -251.759,Z 1209.737,A 0.000,B 0.000,C 90.000,E1 312.609} C_DIS
LIN {X -0.056,Y -263.196,Z 1209.719,A 0.000,B 0.000,C 90.000,E1 309.358} C_DIS
LIN {X 0.107,Y -274.451,Z 1209.703,A 0.000,B 0.000,C 90.000,E1 306.503} C_DIS
LIN {X 0.030,Y -288.847,Z 1209.686,A 0.000,B 0.000,C 90.000,E1 303.420} C_DIS
LIN {X -0.006,Y -305.069,Z 1209.669,A 0.000,B 0.000,C 90.000,E1 300.413} C_DIS
LIN {X 0.131,Y -313.274,Z 1209.662,A 0.000,B 0.000,C 90.000,E1 299.077} C_DIS
LIN {X -0.065,Y -322.435,Z 1209.655,A 0.000,B 0.000,C 90.000,E1 297.820} C_DIS
LIN {X 0.043,Y -334.862,Z 1209.646,A 0.000,B 0.000,C 90.000,E1 296.232} C_DIS
LIN {X 0.205,Y -350.815,Z 1209.636,A 0.000,B 0.000,C 90.000,E1 294.387} C_DIS
LIN {X -0.006,Y -369.002,Z 1209.625,A 0.000,B 0.000,C 90.000,E1 292.461} C_DIS
LIN {X -0.060,Y -387.709,Z 1209.614,A 0.000,B 0.000,C 90.000,E1 290.556} C_DIS
LIN {X 0.095,Y -400.811,Z 1209.607,A 0.000,B 0.000,C 90.000,E1 289.214} C_DIS
LIN {X -0.109,Y -413.857,Z 1209.599,A 0.000,B 0.000,C 90.000,E1 287.928} C_DIS
LIN {X 0.040,Y -423.840,Z 1209.594,A 0.000,B 0.000,C 90.000,E1 286.858} C_DIS
LIN {X -0.169,Y -431.000,Z 1209.589,A 0.000,B 0.000,C 90.000,E1 286.079} C_DIS
LIN {X 0.054,Y -437.621,Z 1209.585,A 0.000,B 0.000,C 90.000,E1 285.245} C_DIS
LIN {X -0.192,Y -443.602,Z 1209.580,A 0.000,B 0.000,C 90.000,E1 284.481} C_DIS
LIN {X 0.150,Y -449.017,Z 1209.576,A 0.000,B 0.000,C 90.000,E1 283.647} C_DIS
LIN {X 0.004,Y -453.783,Z 1209.572,A 0.000,B 0.000,C 90.000,E1 282.883} C_DIS
LIN {X -0.106,Y -457.798,Z 1209.567,A 0.000,B 0.000,C 90.000,E1 282.119} C_DIS
LIN {X -0.009,Y -460.100,Z 1209.564,A 0.000,B 0.000,C 90.000,E1 281.591} C_DIS
LIN {X 0.012,Y -462.139,Z 1209.562,A 0.000,B 0.000,C 90.000,E1 281.074} C_DIS
LIN {X 0.132,Y -463.884,Z 1209.559,A 0.000,B 0.000,C 90.000,E1 280.546} C_DIS
LIN {X -0.197,Y -465.398,Z 1209.556,A 0.000,B 0.000,C 90.000,E1 280.074} C_DIS
LIN {X -0.139,Y -466.625,Z 1209.553,A 0.000,B 0.000,C 90.000,E1 279.557} C_DIS
LIN {X 0.005,Y -467.584,Z 1209.550,A 0.000,B 0.000,C 90.000,E1 279.029} C_DIS
LIN {X 0.084,Y -468.265,Z 1209.547,A 0.000,B 0.000,C 90.000,E1 278.511} C_DIS
LIN {X 0.170,Y -468.740,Z 1209.545,A 0.000,B 0.000,C 90.000,E1 277.992} C_DIS
LIN {X -0.202,Y -468.925,Z 1209.542,A 0.000,B 0.000,C 90.000,E1 277.530} C_DIS
LIN {X -0.049,Y -468.780,Z 1209.539,A 0.000,B 0.000,C 90.000,E1 277.004} C_DIS
LIN {X 0.045,Y -468.243,Z 1209.536,A 0.000,B 0.000,C 90.000,E1 276.486} C_DIS
LIN {X 0.138,Y -467.317,Z 1209.533,A 0.000,B 0.000,C 90.000,E1 275.967} C_DIS
LIN {X 0.183,Y -465.975,Z 1209.530,A 0.000,B 0.000,C 90.000,E1 275.454} C_DIS
LIN {X -0.194,Y -464.160,Z 1209.528,A 0.000,B 0.000,C 90.000,E1 274.992} C_DIS
LIN {X -0.116,Y -461.861,Z 1209.525,A 0.000,B 0.000,C 90.000,E1 274.473} C_DIS
LIN {X -0.058,Y -458.884,Z 1209.522,A 0.000,B 0.000,C 90.000,E1 273.955} C_DIS
LIN {X -0.046,Y -455.091,Z 1209.519,A 0.000,B 0.000,C 90.000,E1 273.440} C_DIS
LIN {X 0.177,Y -452.831,Z 1209.518,A 0.000,B 0.000,C 90.000,E1 273.154} C_DIS
LIN {X -0.195,Y -447.459,Z 1209.515,A 0.000,B 0.000,C 90.000,E1 272.694} C_DIS
LIN {X 0.084,Y -444.263,Z 1209.513,A 0.000,B 0.000,C 90.000,E1 272.407} C_DIS
LIN {X -0.124,Y -437.738,Z 1209.511,A 0.000,B 0.000,C 90.000,E1 272.007} C_DIS
LIN {X -0.168,Y -434.384,Z 1209.510,A 0.000,B 0.000,C 90.000,E1 271.833} C_DIS
LIN {X 0.017,Y -427.001,Z 1209.508,A 0.000,B 0.000,C 90.000,E1 271.489} C_DIS
LIN {X -0.201,Y -416.396,Z 1209.506,A 0.000,B 0.000,C 90.000,E1 271.146} C_DIS
LIN {X 0.129,Y -406.364,Z 1209.505,A 0.000,B 0.000,C 90.000,E1 270.802} C_DIS
LIN {X 0.098,Y -399.448,Z 1209.504,A 0.000,B 0.000,C 90.000,E1 270.630} C_DIS
LIN {X -0.165,Y -392.278,Z 1209.503,A 0.000,B 0.000,C 90.000,E1 270.516} C_DIS
LIN {X 0.181,Y -379.847,Z 1209.502,A 0.000,B 0.000,C 90.000,E1 270.286} C_DIS
LIN {X 0.102,Y -371.676,Z 1209.501,A 0.000,B 0.000,C 90.000,E1 270.229} C_DIS
LIN {X -0.093,Y -363.769,Z 1209.501,A 0.000,B 0.000,C 90.000,E1 270.229} C_DIS
LIN {X -0.070,Y -181.580,Z 1209.501,A 0.000,B 0.000,C 90.000,E1 270.229} C_DIS
LIN {X -0.043,Y -180.883,Z 1209.473,A 0.000,B 0.000,C 90.000,E1 265.122} C_DIS
LIN {X 0.016,Y -179.003,Z 1209.445,A 0.000,B 0.000,C 90.000,E1 260.038} C_DIS
LIN {X -0.065,Y -178.605,Z 1209.440,A 0.000,B 0.000,C 90.000,E1 259.218} C_DIS
LIN {X 0.004,Y -175.657,Z 1209.412,A 0.000,B 0.000,C 90.000,E1 254.102} C_DIS
LIN {X 0.009,Y -172.375,Z 1209.388,A 0.000,B 0.000,C 90.000,E1 249.826} C_DIS
LIN {X 0.023,Y -171.170,Z 1209.378,A 0.000,B 0.000,C 90.000,E1 248.103} C_DIS
LIN {X 0.067,Y -167.466,Z 1209.354,A 0.000,B 0.000,C 90.000,E1 243.768} C_DIS
LIN {X 0.000,Y -166.863,Z 1209.350,A 0.000,B 0.000,C 90.000,E1 242.922} C_DIS
LIN {X 0.054,Y -162.167,Z 1209.320,A 0.000,B 0.000,C 90.000,E1 237.661} C_DIS
LIN {X -0.025,Y -160.729,Z 1209.311,A 0.000,B 0.000,C 90.000,E1 235.928} C_DIS
LIN {X -0.046,Y -157.532,Z 1209.291,A 0.000,B 0.000,C 90.000,E1 232.396} C_DIS
LIN {X 0.012,Y -155.558,Z 1209.276,A 0.000,B 0.000,C 90.000,E1 229.703} C_DIS
LIN {X -0.055,Y -151.848,Z 1209.251,A 0.000,B 0.000,C 90.000,E1 225.243} C_DIS
LIN {X -0.040,Y -150.068,Z 1209.236,A 0.000,B 0.000,C 90.000,E1 222.528} C_DIS
LIN {X -0.006,Y -146.876,Z 1209.211,A 0.000,B 0.000,C 90.000,E1 217.971} C_DIS
LIN {X -0.017,Y -145.462,Z 1209.196,A 0.000,B 0.000,C 90.000,E1 215.231} C_DIS
LIN {X 0.024,Y -142.876,Z 1209.170,A 0.000,B 0.000,C 90.000,E1 210.620} C_DIS
LIN {X 0.022,Y -141.493,Z 1209.150,A 0.000,B 0.000,C 90.000,E1 206.924} C_DIS
LIN {X 0.007,Y -139.386,Z 1209.114,A 0.000,B 0.000,C 90.000,E1 200.429} C_DIS
LIN {X -0.005,Y -138.842,Z 1209.098,A 0.000,B 0.000,C 90.000,E1 197.638} C_DIS
LIN {X 0.056,Y -138.353,Z 1209.057,A 0.000,B 0.000,C 90.000,E1 190.141} C_DIS
LIN {X 0.051,Y -139.519,Z 1209.005,A 0.000,B 0.000,C 90.000,E1 180.802} C_DIS
LIN {X -0.007,Y -141.179,Z 1208.974,A 0.000,B 0.000,C 90.000,E1 175.241} C_DIS
LIN {X -0.037,Y -142.557,Z 1208.958,A 0.000,B 0.000,C 90.000,E1 172.470} C_DIS
LIN {X 0.030,Y -144.838,Z 1208.932,A 0.000,B 0.000,C 90.000,E1 167.825} C_DIS
LIN {X 0.016,Y -147.461,Z 1208.912,A 0.000,B 0.000,C 90.000,E1 164.157} C_DIS
LIN {X 0.043,Y -150.045,Z 1208.892,A 0.000,B 0.000,C 90.000,E1 160.496} C_DIS
LIN {X 0.048,Y -153.387,Z 1208.872,A 0.000,B 0.000,C 90.000,E1 156.869} C_DIS
LIN {X -0.045,Y -155.918,Z 1208.857,A 0.000,B 0.000,C 90.000,E1 154.204} C_DIS
LIN {X 0.069,Y -159.783,Z 1208.837,A 0.000,B 0.000,C 90.000,E1 150.589} C_DIS
LIN {X -0.083,Y -162.023,Z 1208.827,A 0.000,B 0.000,C 90.000,E1 148.869} C_DIS
LIN {X 0.030,Y -166.217,Z 1208.807,A 0.000,B 0.000,C 90.000,E1 145.308} C_DIS
LIN {X 0.033,Y -171.233,Z 1208.788,A 0.000,B 0.000,C 90.000,E1 141.823} C_DIS
LIN {X -0.044,Y -176.120,Z 1208.769,A 0.000,B 0.000,C 90.000,E1 138.405} C_DIS
LIN {X 0.072,Y -180.385,Z 1208.755,A 0.000,B 0.000,C 90.000,E1 135.810} C_DIS
LIN {X 0.048,Y -185.793,Z 1208.736,A 0.000,B 0.000,C 90.000,E1 132.447} C_DIS
LIN {X -0.019,Y -190.410,Z 1208.722,A 0.000,B 0.000,C 90.000,E1 129.967} C_DIS
LIN {X -0.003,Y -197.734,Z 1208.699,A 0.000,B 0.000,C 90.000,E1 125.851} C_DIS
LIN {X -0.124,Y -201.432,Z 1208.689,A 0.000,B 0.000,C 90.000,E1 123.992} C_DIS
LIN {X 0.205,Y -311.762,Z 1208.689,A 0.000,B 0.000,C 90.000,E1 123.913} C_DIS
LIN {X -0.019,Y -313.894,Z 1208.688,A 0.000,B 0.000,C 90.000,E1 123.913} C_DIS
LIN {X 0.021,Y -318.646,Z 1208.687,A 0.000,B 0.000,C 90.000,E1 123.658} C_DIS
LIN {X -0.029,Y -321.316,Z 1208.686,A 0.000,B 0.000,C 90.000,E1 123.420} C_DIS
LIN {X 0.051,Y -325.040,Z 1208.683,A 0.000,B 0.000,C 90.000,E1 122.880} C_DIS
LIN {X 0.138,Y -326.611,Z 1208.681,A 0.000,B 0.000,C 90.000,E1 122.546} C_DIS
LIN {X -0.040,Y -340.029,Z 1208.662,A 0.000,B 0.000,C 90.000,E1 119.127} C_DIS
LIN {X -0.006,Y -352.457,Z 1208.646,A 0.000,B 0.000,C 90.000,E1 116.360} C_DIS
LIN {X 0.081,Y -366.387,Z 1208.631,A 0.000,B 0.000,C 90.000,E1 113.643} C_DIS
LIN {X 0.160,Y -380.125,Z 1208.618,A 0.000,B 0.000,C 90.000,E1 111.280} C_DIS
LIN {X -0.193,Y -395.241,Z 1208.606,A 0.000,B 0.000,C 90.000,E1 109.033} C_DIS
LIN {X 0.204,Y -411.840,Z 1208.593,A 0.000,B 0.000,C 90.000,E1 106.732} C_DIS
LIN {X -0.144,Y -430.041,Z 1208.581,A 0.000,B 0.000,C 90.000,E1 104.592} C_DIS
LIN {X -0.087,Y -449.735,Z 1208.569,A 0.000,B 0.000,C 90.000,E1 102.479} C_DIS
LIN {X -0.084,Y -472.455,Z 1208.557,A 0.000,B 0.000,C 90.000,E1 100.310} C_DIS
LIN {X -0.036,Y -474.262,Z 1208.556,A 0.000,B 0.000,C 90.000,E1 100.074} C_DIS
LIN {X -0.257,Y -475.770,Z 1208.555,A 0.000,B 0.000,C 90.000,E1 99.849} C_DIS
LIN {X 0.073,Y -476.897,Z 1208.553,A 0.000,B 0.000,C 90.000,E1 99.557} C_DIS
LIN {X -0.190,Y -478.241,Z 1208.550,A 0.000,B 0.000,C 90.000,E1 99.086} C_DIS
LIN {X -0.052,Y -478.562,Z 1208.548,A 0.000,B 0.000,C 90.000,E1 98.568} C_DIS
LIN {X 0.097,Y -477.912,Z 1208.545,A 0.000,B 0.000,C 90.000,E1 98.049} C_DIS
LIN {X -0.222,Y -476.188,Z 1208.542,A 0.000,B 0.000,C 90.000,E1 97.587} C_DIS
LIN {X 0.119,Y -474.827,Z 1208.541,A 0.000,B 0.000,C 90.000,E1 97.296} C_DIS
LIN {X 0.081,Y -460.296,Z 1208.529,A 0.000,B 0.000,C 90.000,E1 95.277} C_DIS
LIN {X -0.190,Y -441.022,Z 1208.514,A 0.000,B 0.000,C 90.000,E1 92.465} C_DIS
LIN {X -0.201,Y -423.361,Z 1208.497,A 0.000,B 0.000,C 90.000,E1 89.542} C_DIS
LIN {X -0.169,Y -411.545,Z 1208.485,A 0.000,B 0.000,C 90.000,E1 87.364} C_DIS
LIN {X 0.034,Y -399.985,Z 1208.473,A 0.000,B 0.000,C 90.000,E1 85.122} C_DIS
LIN {X -0.052,Y -389.759,Z 1208.462,A 0.000,B 0.000,C 90.000,E1 83.166} C_DIS
LIN {X 0.118,Y -379.497,Z 1208.451,A 0.000,B 0.000,C 90.000,E1 81.141} C_DIS
LIN {X 0.132,Y -371.999,Z 1208.443,A 0.000,B 0.000,C 90.000,E1 79.690} C_DIS
LIN {X 0.075,Y -362.659,Z 1208.433,A 0.000,B 0.000,C 90.000,E1 77.937} C_DIS
LIN {X -0.126,Y -351.510,Z 1208.421,A 0.000,B 0.000,C 90.000,E1 75.880} C_DIS
LIN {X -0.042,Y -340.299,Z 1208.410,A 0.000,B 0.000,C 90.000,E1 73.740} C_DIS
LIN {X 0.141,Y -326.016,Z 1208.394,A 0.000,B 0.000,C 90.000,E1 70.913} C_DIS
LIN {X -0.153,Y -312.354,Z 1208.378,A 0.000,B 0.000,C 90.000,E1 68.103} C_DIS
LIN {X 0.106,Y -298.145,Z 1208.360,A 0.000,B 0.000,C 90.000,E1 64.793} C_DIS
LIN {X -0.064,Y -286.320,Z 1208.343,A 0.000,B 0.000,C 90.000,E1 61.820} C_DIS
LIN {X -0.082,Y -273.934,Z 1208.324,A 0.000,B 0.000,C 90.000,E1 58.408} C_DIS
LIN {X -0.001,Y -262.519,Z 1208.305,A 0.000,B 0.000,C 90.000,E1 54.895} C_DIS
LIN {X -0.038,Y -252.969,Z 1208.287,A 0.000,B 0.000,C 90.000,E1 51.698} C_DIS
LIN {X -0.094,Y -242.923,Z 1208.267,A 0.000,B 0.000,C 90.000,E1 48.081} C_DIS
LIN {X 0.087,Y -235.318,Z 1208.251,A 0.000,B 0.000,C 90.000,E1 45.081} C_DIS
LIN {X -0.044,Y -226.210,Z 1208.230,A 0.000,B 0.000,C 90.000,E1 41.353} C_DIS
LIN {X -0.074,Y -219.410,Z 1208.213,A 0.000,B 0.000,C 90.000,E1 38.302} C_DIS
LIN {X -0.017,Y -213.376,Z 1208.195,A 0.000,B 0.000,C 90.000,E1 35.185} C_DIS
LIN {X -0.042,Y -206.742,Z 1208.174,A 0.000,B 0.000,C 90.000,E1 31.258} C_DIS
LIN {X 0.005,Y -201.052,Z 1208.151,A 0.000,B 0.000,C 90.000,E1 27.257} C_DIS
LIN {X 0.050,Y -196.026,Z 1208.129,A 0.000,B 0.000,C 90.000,E1 23.206} C_DIS
LIN {X -0.007,Y -191.846,Z 1208.106,A 0.000,B 0.000,C 90.000,E1 19.141} C_DIS
LIN {X 0.017,Y -187.937,Z 1208.079,A 0.000,B 0.000,C 90.000,E1 14.189} C_DIS
LIN {X -0.072,Y -185.064,Z 1208.047,A 0.000,B 0.000,C 90.000,E1 8.398} C_DIS
LIN {X 0.094,Y -186.034,Z 1207.970,A 0.000,B 0.000,C 90.000,E1 354.489} C_DIS
LIN {X 0.053,Y -188.969,Z 1207.942,A 0.000,B 0.000,C 90.000,E1 349.511} C_DIS
LIN {X -0.044,Y -192.484,Z 1207.919,A 0.000,B 0.000,C 90.000,E1 345.408} C_DIS
LIN {X 0.076,Y -196.889,Z 1207.896,A 0.000,B 0.000,C 90.000,E1 341.275} C_DIS
LIN {X 0.037,Y -202.040,Z 1207.874,A 0.000,B 0.000,C 90.000,E1 337.230} C_DIS
LIN {X -0.087,Y -207.920,Z 1207.851,A 0.000,B 0.000,C 90.000,E1 333.256} C_DIS
LIN {X -0.060,Y -212.941,Z 1207.834,A 0.000,B 0.000,C 90.000,E1 330.078} C_DIS
LIN {X 0.044,Y -219.626,Z 1207.812,A 0.000,B 0.000,C 90.000,E1 326.135} C_DIS
LIN {X 0.069,Y -227.030,Z 1207.791,A 0.000,B 0.000,C 90.000,E1 322.271} C_DIS
LIN {X 0.019,Y -235.288,Z 1207.769,A 0.000,B 0.000,C 90.000,E1 318.485} C_DIS
LIN {X 0.032,Y -243.890,Z 1207.751,A 0.000,B 0.000,C 90.000,E1 315.121} C_DIS
LIN {X 0.140,Y -251.680,Z 1207.736,A 0.000,B 0.000,C 90.000,E1 312.528} C_DIS
LIN {X 0.138,Y -261.839,Z 1207.720,A 0.000,B 0.000,C 90.000,E1 309.644} C_DIS
LIN {X -0.112,Y -272.961,Z 1207.705,A 0.000,B 0.000,C 90.000,E1 306.870} C_DIS
LIN {X 0.040,Y -285.515,Z 1207.689,A 0.000,B 0.000,C 90.000,E1 304.072} C_DIS
LIN {X -0.036,Y -297.729,Z 1207.676,A 0.000,B 0.000,C 90.000,E1 301.720} C_DIS
LIN {X 0.021,Y -307.132,Z 1207.667,A 0.000,B 0.000,C 90.000,E1 300.050} C_DIS
LIN {X 0.026,Y -315.592,Z 1207.660,A 0.000,B 0.000,C 90.000,E1 298.743} C_DIS
LIN {X -0.009,Y -324.890,Z 1207.653,A 0.000,B 0.000,C 90.000,E1 297.462} C_DIS
LIN {X 0.099,Y -335.005,Z 1207.646,A 0.000,B 0.000,C 90.000,E1 296.181} C_DIS
LIN {X 0.067,Y -350.790,Z 1207.635,A 0.000,B 0.000,C 90.000,E1 294.387} C_DIS
LIN {X -0.118,Y -368.962,Z 1207.625,A 0.000,B 0.000,C 90.000,E1 292.461} C_DIS
LIN {X -0.152,Y -390.277,Z 1207.613,A 0.000,B 0.000,C 90.000,E1 290.301} C_DIS
LIN {X 0.219,Y -403.055,Z 1207.605,A 0.000,B 0.000,C 90.000,E1 288.960} C_DIS
LIN {X -0.081,Y -416.092,Z 1207.598,A 0.000,B 0.000,C 90.000,E1 287.692} C_DIS
LIN {X -0.167,Y -423.565,Z 1207.594,A 0.000,B 0.000,C 90.000,E1 286.913} C_DIS
LIN {X 0.033,Y -430.737,Z 1207.589,A 0.000,B 0.000,C 90.000,E1 286.079} C_DIS
LIN {X -0.165,Y -437.384,Z 1207.585,A 0.000,B 0.000,C 90.000,E1 285.300} C_DIS
LIN {X 0.010,Y -443.398,Z 1207.580,A 0.000,B 0.000,C 90.000,E1 284.481} C_DIS
LIN {X -0.082,Y -448.875,Z 1207.576,A 0.000,B 0.000,C 90.000,E1 283.703} C_DIS
LIN {X 0.209,Y -453.618,Z 1207.572,A 0.000,B 0.000,C 90.000,E1 282.883} C_DIS
LIN {X 0.099,Y -457.680,Z 1207.567,A 0.000,B 0.000,C 90.000,E1 282.119} C_DIS
LIN {X -0.066,Y -461.035,Z 1207.563,A 0.000,B 0.000,C 90.000,E1 281.366} C_DIS
LIN {X -0.112,Y -463.823,Z 1207.559,A 0.000,B 0.000,C 90.000,E1 280.602} C_DIS
LIN {X 0.015,Y -465.323,Z 1207.556,A 0.000,B 0.000,C 90.000,E1 280.074} C_DIS
LIN {X 0.073,Y -466.534,Z 1207.553,A 0.000,B 0.000,C 90.000,E1 279.557} C_DIS
LIN {X 0.217,Y -467.526,Z 1207.550,A 0.000,B 0.000,C 90.000,E1 279.029} C_DIS
LIN {X -0.167,Y -468.240,Z 1207.547,A 0.000,B 0.000,C 90.000,E1 278.568} C_DIS
LIN {X -0.082,Y -468.733,Z 1207.545,A 0.000,B 0.000,C 90.000,E1 278.049} C_DIS
LIN {X 0.009,Y -468.937,Z 1207.542,A 0.000,B 0.000,C 90.000,E1 277.530} C_DIS
LIN {X 0.106,Y -468.854,Z 1207.539,A 0.000,B 0.000,C 90.000,E1 277.011} C_DIS
LIN {X 0.256,Y -468.413,Z 1207.536,A 0.000,B 0.000,C 90.000,E1 276.486} C_DIS
LIN {X -0.115,Y -467.547,Z 1207.533,A 0.000,B 0.000,C 90.000,E1 276.024} C_DIS
LIN {X -0.069,Y -466.261,Z 1207.531,A 0.000,B 0.000,C 90.000,E1 275.511} C_DIS
LIN {X 0.018,Y -464.500,Z 1207.528,A 0.000,B 0.000,C 90.000,E1 274.992} C_DIS
LIN {X 0.097,Y -462.229,Z 1207.525,A 0.000,B 0.000,C 90.000,E1 274.473} C_DIS
LIN {X 0.155,Y -459.326,Z 1207.522,A 0.000,B 0.000,C 90.000,E1 273.955} C_DIS
LIN {X 0.167,Y -455.628,Z 1207.519,A 0.000,B 0.000,C 90.000,E1 273.440} C_DIS
LIN {X 0.189,Y -450.892,Z 1207.516,A 0.000,B 0.000,C 90.000,E1 272.922} C_DIS
LIN {X -0.018,Y -448.107,Z 1207.515,A 0.000,B 0.000,C 90.000,E1 272.694} C_DIS
LIN {X -0.113,Y -441.848,Z 1207.512,A 0.000,B 0.000,C 90.000,E1 272.236} C_DIS
LIN {X -0.006,Y -438.415,Z 1207.511,A 0.000,B 0.000,C 90.000,E1 272.007} C_DIS
LIN {X -0.127,Y -431.253,Z 1207.509,A 0.000,B 0.000,C 90.000,E1 271.661} C_DIS
LIN {X -0.133,Y -420.744,Z 1207.507,A 0.000,B 0.000,C 90.000,E1 271.260} C_DIS
LIN {X 0.073,Y -410.606,Z 1207.505,A 0.000,B 0.000,C 90.000,E1 270.917} C_DIS
LIN {X 0.173,Y -400.538,Z 1207.504,A 0.000,B 0.000,C 90.000,E1 270.630} C_DIS
LIN {X -0.123,Y -393.294,Z 1207.503,A 0.000,B 0.000,C 90.000,E1 270.516} C_DIS
LIN {X 0.183,Y -381.281,Z 1207.502,A 0.000,B 0.000,C 90.000,E1 270.286} C_DIS
LIN {X 0.085,Y -373.809,Z 1207.501,A 0.000,B 0.000,C 90.000,E1 270.229} C_DIS
LIN {X -0.172,Y -365.424,Z 1207.501,A 0.000,B 0.000,C 90.000,E1 270.229} C_DIS
LIN {X 0.071,Y -181.580,Z 1207.501,A 0.000,B 0.000,C 90.000,E1 270.172} C_DIS
LIN {X -0.065,Y -180.882,Z 1207.473,A 0.000,B 0.000,C 90.000,E1 265.122} C_DIS
LIN {X -0.006,Y -179.002,Z 1207.445,A 0.000,B 0.000,C 90.000,E1 260.038} C_DIS
LIN {X 0.088,Y -178.599,Z 1207.440,A 0.000,B 0.000,C 90.000,E1 259.162} C_DIS
LIN {X -0.019,Y -175.652,Z 1207.412,A 0.000,B 0.000,C 90.000,E1 254.102} C_DIS
LIN {X -0.013,Y -172.370,Z 1207.388,A 0.000,B 0.000,C 90.000,E1 249.826} C_DIS
LIN {X 0.001,Y -171.163,Z 1207.378,A 0.000,B 0.000,C 90.000,E1 248.103} C_DIS
LIN {X 0.046,Y -167.461,Z 1207.354,A 0.000,B 0.000,C 90.000,E1 243.768} C_DIS
LIN {X -0.021,Y -166.857,Z 1207.349,A 0.000,B 0.000,C 90.000,E1 242.922} C_DIS
LIN {X 0.043,Y -162.843,Z 1207.325,A 0.000,B 0.000,C 90.000,E1 238.535} C_DIS
LIN {X 0.018,Y -161.526,Z 1207.316,A 0.000,B 0.000,C 90.000,E1 236.786} C_DIS
LIN {X 0.059,Y -157.526,Z 1207.291,A 0.000,B 0.000,C 90.000,E1 232.351} C_DIS
LIN {X -0.009,Y -155.551,Z 1207.276,A 0.000,B 0.000,C 90.000,E1 229.703} C_DIS
LIN {X -0.074,Y -151.842,Z 1207.251,A 0.000,B 0.000,C 90.000,E1 225.243} C_DIS
LIN {X -0.060,Y -150.062,Z 1207.236,A 0.000,B 0.000,C 90.000,E1 222.528} C_DIS
LIN {X -0.025,Y -146.871,Z 1207.211,A 0.000,B 0.000,C 90.000,E1 217.971} C_DIS
LIN {X -0.036,Y -145.456,Z 1207.196,A 0.000,B 0.000,C 90.000,E1 215.231} C_DIS
LIN {X 0.077,Y -142.872,Z 1207.170,A 0.000,B 0.000,C 90.000,E1 210.590} C_DIS
LIN {X 0.002,Y -141.490,Z 1207.150,A 0.000,B 0.000,C 90.000,E1 206.924} C_DIS
LIN {X -0.013,Y -139.385,Z 1207.114,A 0.000,B 0.000,C 90.000,E1 200.429} C_DIS
LIN {X -0.023,Y -138.841,Z 1207.098,A 0.000,B 0.000,C 90.000,E1 197.638} C_DIS
LIN {X 0.037,Y -138.354,Z 1207.056,A 0.000,B 0.000,C 90.000,E1 190.141} C_DIS
LIN {X 0.032,Y -139.520,Z 1207.005,A 0.000,B 0.000,C 90.000,E1 180.802} C_DIS
LIN {X -0.027,Y -141.182,Z 1206.974,A 0.000,B 0.000,C 90.000,E1 175.241} C_DIS
LIN {X -0.056,Y -142.561,Z 1206.958,A 0.000,B 0.000,C 90.000,E1 172.470} C_DIS
LIN {X 0.010,Y -144.843,Z 1206.932,A 0.000,B 0.000,C 90.000,E1 167.825} C_DIS
LIN {X -0.004,Y -147.467,Z 1206.912,A 0.000,B 0.000,C 90.000,E1 164.157} C_DIS
LIN {X 0.023,Y -150.051,Z 1206.892,A 0.000,B 0.000,C 90.000,E1 160.496} C_DIS
LIN {X 0.028,Y -153.395,Z 1206.872,A 0.000,B 0.000,C 90.000,E1 156.869} C_DIS
LIN {X 0.074,Y -155.925,Z 1206.857,A 0.000,B 0.000,C 90.000,E1 154.152} C_DIS
LIN {X 0.049,Y -159.792,Z 1206.837,A 0.000,B 0.000,C 90.000,E1 150.589} C_DIS
LIN {X 0.034,Y -162.032,Z 1206.827,A 0.000,B 0.000,C 90.000,E1 148.820} C_DIS
LIN {X 0.009,Y -166.226,Z 1206.807,A 0.000,B 0.000,C 90.000,E1 145.308} C_DIS
LIN {X 0.010,Y -171.243,Z 1206.788,A 0.000,B 0.000,C 90.000,E1 141.823} C_DIS
LIN {X -0.067,Y -176.132,Z 1206.769,A 0.000,B 0.000,C 90.000,E1 138.405} C_DIS
LIN {X 0.049,Y -180.397,Z 1206.755,A 0.000,B 0.000,C 90.000,E1 135.810} C_DIS
LIN {X 0.026,Y -185.805,Z 1206.736,A 0.000,B 0.000,C 90.000,E1 132.447} C_DIS
LIN {X 0.081,Y -190.423,Z 1206.722,A 0.000,B 0.000,C 90.000,E1 129.930} C_DIS
LIN {X -0.028,Y -197.748,Z 1206.699,A 0.000,B 0.000,C 90.000,E1 125.851} C_DIS
LIN {X 0.055,Y -201.481,Z 1206.688,A 0.000,B 0.000,C 90.000,E1 123.913} C_DIS
LIN {X 0.037,Y -311.519,Z 1206.688,A 0.000,B 0.000,C 90.000,E1 123.913} C_DIS
LIN {X -0.057,Y -312.896,Z 1206.688,A 0.000,B 0.000,C 90.000,E1 123.913} C_DIS
LIN {X -0.018,Y -318.399,Z 1206.687,A 0.000,B 0.000,C 90.000,E1 123.658} C_DIS
LIN {X -0.067,Y -321.178,Z 1206.686,A 0.000,B 0.000,C 90.000,E1 123.420} C_DIS
LIN {X 0.106,Y -324.901,Z 1206.683,A 0.000,B 0.000,C 90.000,E1 122.880} C_DIS
LIN {X 0.194,Y -326.522,Z 1206.681,A 0.000,B 0.000,C 90.000,E1 122.546} C_DIS
LIN {X 0.015,Y -339.970,Z 1206.662,A 0.000,B 0.000,C 90.000,E1 119.127} C_DIS
LIN {X 0.048,Y -352.392,Z 1206.646,A 0.000,B 0.000,C 90.000,E1 116.360} C_DIS
LIN {X 0.136,Y -366.316,Z 1206.631,A 0.000,B 0.000,C 90.000,E1 113.643} C_DIS
LIN {X 0.215,Y -380.049,Z 1206.618,A 0.000,B 0.000,C 90.000,E1 111.280} C_DIS
LIN {X -0.138,Y -395.159,Z 1206.606,A 0.000,B 0.000,C 90.000,E1 109.033} C_DIS
LIN {X -0.254,Y -411.753,Z 1206.593,A 0.000,B 0.000,C 90.000,E1 106.804} C_DIS
LIN {X -0.089,Y -429.947,Z 1206.581,A 0.000,B 0.000,C 90.000,E1 104.592} C_DIS
LIN {X -0.033,Y -449.639,Z 1206.569,A 0.000,B 0.000,C 90.000,E1 102.479} C_DIS
LIN {X -0.034,Y -472.356,Z 1206.557,A 0.000,B 0.000,C 90.000,E1 100.310} C_DIS
LIN {X 0.015,Y -474.163,Z 1206.556,A 0.000,B 0.000,C 90.000,E1 100.074} C_DIS
LIN {X -0.207,Y -475.672,Z 1206.555,A 0.000,B 0.000,C 90.000,E1 99.849} C_DIS
LIN {X 0.124,Y -476.797,Z 1206.553,A 0.000,B 0.000,C 90.000,E1 99.557} C_DIS
LIN {X -0.215,Y -478.138,Z 1206.550,A 0.000,B 0.000,C 90.000,E1 99.095} C_DIS
LIN {X -0.003,Y -478.457,Z 1206.548,A 0.000,B 0.000,C 90.000,E1 98.568} C_DIS
LIN {X 0.147,Y -477.805,Z 1206.545,A 0.000,B 0.000,C 90.000,E1 98.049} C_DIS
LIN {X -0.174,Y -476.081,Z 1206.542,A 0.000,B 0.000,C 90.000,E1 97.587} C_DIS
LIN {X 0.166,Y -474.719,Z 1206.541,A 0.000,B 0.000,C 90.000,E1 97.296} C_DIS
LIN {X -0.093,Y -458.391,Z 1206.528,A 0.000,B 0.000,C 90.000,E1 95.049} C_DIS
LIN {X -0.151,Y -440.904,Z 1206.514,A 0.000,B 0.000,C 90.000,E1 92.465} C_DIS
LIN {X -0.168,Y -423.259,Z 1206.497,A 0.000,B 0.000,C 90.000,E1 89.542} C_DIS
LIN {X -0.140,Y -411.448,Z 1206.485,A 0.000,B 0.000,C 90.000,E1 87.364} C_DIS
LIN {X 0.061,Y -399.873,Z 1206.473,A 0.000,B 0.000,C 90.000,E1 85.122} C_DIS
LIN {X -0.027,Y -389.652,Z 1206.462,A 0.000,B 0.000,C 90.000,E1 83.166} C_DIS
LIN {X 0.115,Y -380.869,Z 1206.453,A 0.000,B 0.000,C 90.000,E1 81.432} C_DIS
LIN {X 0.151,Y -371.881,Z 1206.443,A 0.000,B 0.000,C 90.000,E1 79.690} C_DIS
LIN {X 0.092,Y -362.549,Z 1206.433,A 0.000,B 0.000,C 90.000,E1 77.937} C_DIS
LIN {X -0.112,Y -351.398,Z 1206.422,A 0.000,B 0.000,C 90.000,E1 75.880} C_DIS
LIN {X -0.031,Y -340.179,Z 1206.410,A 0.000,B 0.000,C 90.000,E1 73.740} C_DIS
LIN {X 0.148,Y -325.902,Z 1206.394,A 0.000,B 0.000,C 90.000,E1 70.913} C_DIS
LIN {X -0.150,Y -312.231,Z 1206.378,A 0.000,B 0.000,C 90.000,E1 68.103} C_DIS
LIN {X 0.106,Y -298.026,Z 1206.360,A 0.000,B 0.000,C 90.000,E1 64.793} C_DIS
LIN {X -0.067,Y -286.185,Z 1206.343,A 0.000,B 0.000,C 90.000,E1 61.820} C_DIS
LIN {X -0.089,Y -273.808,Z 1206.324,A 0.000,B 0.000,C 90.000,E1 58.408} C_DIS
LIN {X -0.012,Y -262.356,Z 1206.305,A 0.000,B 0.000,C 90.000,E1 54.895} C_DIS
LIN {X -0.053,Y -252.778,Z 1206.287,A 0.000,B 0.000,C 90.000,E1 51.698} C_DIS
LIN {X -0.114,Y -242.682,Z 1206.267,A 0.000,B 0.000,C 90.000,E1 48.081} C_DIS
LIN {X 0.061,Y -235.055,Z 1206.250,A 0.000,B 0.000,C 90.000,E1 45.081} C_DIS
LIN {X 0.093,Y -225.895,Z 1206.230,A 0.000,B 0.000,C 90.000,E1 41.310} C_DIS
LIN {X 0.058,Y -219.135,Z 1206.213,A 0.000,B 0.000,C 90.000,E1 38.257} C_DIS
LIN {X -0.062,Y -213.129,Z 1206.195,A 0.000,B 0.000,C 90.000,E1 35.185} C_DIS
LIN {X -0.094,Y -206.508,Z 1206.173,A 0.000,B 0.000,C 90.000,E1 31.258} C_DIS
LIN {X -0.053,Y -200.795,Z 1206.151,A 0.000,B 0.000,C 90.000,E1 27.257} C_DIS
LIN {X -0.014,Y -195.756,Z 1206.129,A 0.000,B 0.000,C 90.000,E1 23.206} C_DIS
LIN {X -0.077,Y -191.548,Z 1206.106,A 0.000,B 0.000,C 90.000,E1 19.141} C_DIS
LIN {X -0.018,Y -187.622,Z 1206.079,A 0.000,B 0.000,C 90.000,E1 14.175} C_DIS
LIN {X 0.018,Y -184.748,Z 1206.046,A 0.000,B 0.000,C 90.000,E1 8.341} C_DIS
LIN {X 0.082,Y -185.689,Z 1205.969,A 0.000,B 0.000,C 90.000,E1 354.489} C_DIS
LIN {X 0.028,Y -188.631,Z 1205.942,A 0.000,B 0.000,C 90.000,E1 349.511} C_DIS
LIN {X -0.044,Y -192.960,Z 1205.914,A 0.000,B 0.000,C 90.000,E1 344.574} C_DIS
LIN {X -0.031,Y -197.581,Z 1205.891,A 0.000,B 0.000,C 90.000,E1 340.477} C_DIS
LIN {X 0.029,Y -202.870,Z 1205.869,A 0.000,B 0.000,C 90.000,E1 336.410} C_DIS
LIN {X 0.025,Y -208.886,Z 1205.847,A 0.000,B 0.000,C 90.000,E1 332.410} C_DIS
LIN {X 0.001,Y -213.951,Z 1205.829,A 0.000,B 0.000,C 90.000,E1 329.253} C_DIS
LIN {X 0.021,Y -220.782,Z 1205.807,A 0.000,B 0.000,C 90.000,E1 325.341} C_DIS
LIN {X 0.023,Y -228.360,Z 1205.786,A 0.000,B 0.000,C 90.000,E1 321.492} C_DIS
LIN {X -0.093,Y -235.062,Z 1205.769,A 0.000,B 0.000,C 90.000,E1 318.485} C_DIS
LIN {X -0.069,Y -242.713,Z 1205.753,A 0.000,B 0.000,C 90.000,E1 315.486} C_DIS
LIN {X 0.007,Y -250.410,Z 1205.738,A 0.000,B 0.000,C 90.000,E1 312.894} C_DIS
LIN {X -0.039,Y -260.446,Z 1205.722,A 0.000,B 0.000,C 90.000,E1 310.011} C_DIS
LIN {X 0.127,Y -272.957,Z 1205.705,A 0.000,B 0.000,C 90.000,E1 306.790} C_DIS
LIN {X 0.050,Y -285.541,Z 1205.689,A 0.000,B 0.000,C 90.000,E1 304.040} C_DIS
LIN {X 0.061,Y -297.755,Z 1205.676,A 0.000,B 0.000,C 90.000,E1 301.671} C_DIS
LIN {X 0.127,Y -307.270,Z 1205.667,A 0.000,B 0.000,C 90.000,E1 300.001} C_DIS
LIN {X -0.079,Y -317.958,Z 1205.658,A 0.000,B 0.000,C 90.000,E1 298.409} C_DIS
LIN {X -0.089,Y -327.413,Z 1205.651,A 0.000,B 0.000,C 90.000,E1 297.129} C_DIS
LIN {X 0.188,Y -337.515,Z 1205.644,A 0.000,B 0.000,C 90.000,E1 295.848} C_DIS
LIN {X 0.076,Y -350.554,Z 1205.635,A 0.000,B 0.000,C 90.000,E1 294.387} C_DIS
LIN {X -0.122,Y -368.763,Z 1205.625,A 0.000,B 0.000,C 90.000,E1 292.461} C_DIS
LIN {X -0.120,Y -390.097,Z 1205.613,A 0.000,B 0.000,C 90.000,E1 290.301} C_DIS
LIN {X -0.163,Y -400.481,Z 1205.607,A 0.000,B 0.000,C 90.000,E1 289.268} C_DIS
LIN {X 0.106,Y -413.264,Z 1205.600,A 0.000,B 0.000,C 90.000,E1 287.946} C_DIS
LIN {X 0.028,Y -420.928,Z 1205.595,A 0.000,B 0.000,C 90.000,E1 287.166} C_DIS
LIN {X -0.064,Y -428.260,Z 1205.591,A 0.000,B 0.000,C 90.000,E1 286.370} C_DIS
LIN {X 0.022,Y -435.149,Z 1205.586,A 0.000,B 0.000,C 90.000,E1 285.552} C_DIS
LIN {X -0.137,Y -441.385,Z 1205.582,A 0.000,B 0.000,C 90.000,E1 284.773} C_DIS
LIN {X 0.082,Y -447.038,Z 1205.578,A 0.000,B 0.000,C 90.000,E1 283.953} C_DIS
LIN {X 0.021,Y -452.043,Z 1205.573,A 0.000,B 0.000,C 90.000,E1 283.175} C_DIS
LIN {X -0.100,Y -456.348,Z 1205.569,A 0.000,B 0.000,C 90.000,E1 282.411} C_DIS
LIN {X 0.166,Y -459.983,Z 1205.565,A 0.000,B 0.000,C 90.000,E1 281.602} C_DIS
LIN {X -0.173,Y -462.027,Z 1205.562,A 0.000,B 0.000,C 90.000,E1 281.130} C_DIS
LIN {X -0.049,Y -463.800,Z 1205.559,A 0.000,B 0.000,C 90.000,E1 280.602} C_DIS
LIN {X 0.079,Y -465.290,Z 1205.556,A 0.000,B 0.000,C 90.000,E1 280.074} C_DIS
LIN {X 0.137,Y -466.501,Z 1205.553,A 0.000,B 0.000,C 90.000,E1 279.557} C_DIS
LIN {X -0.180,Y -467.492,Z 1205.550,A 0.000,B 0.000,C 90.000,E1 279.086} C_DIS
LIN {X -0.104,Y -468.231,Z 1205.547,A 0.000,B 0.000,C 90.000,E1 278.568} C_DIS
LIN {X -0.019,Y -468.727,Z 1205.545,A 0.000,B 0.000,C 90.000,E1 278.049} C_DIS
LIN {X 0.073,Y -468.964,Z 1205.542,A 0.000,B 0.000,C 90.000,E1 277.530} C_DIS
LIN {X 0.169,Y -468.957,Z 1205.539,A 0.000,B 0.000,C 90.000,E1 277.011} C_DIS
LIN {X -0.145,Y -468.561,Z 1205.536,A 0.000,B 0.000,C 90.000,E1 276.543} C_DIS
LIN {X -0.100,Y -467.728,Z 1205.533,A 0.000,B 0.000,C 90.000,E1 276.030} C_DIS
LIN {X -0.005,Y -466.448,Z 1205.531,A 0.000,B 0.000,C 90.000,E1 275.511} C_DIS
LIN {X 0.084,Y -464.718,Z 1205.528,A 0.000,B 0.000,C 90.000,E1 274.992} C_DIS
LIN {X 0.163,Y -462.499,Z 1205.525,A 0.000,B 0.000,C 90.000,E1 274.473} C_DIS
LIN {X 0.223,Y -459.629,Z 1205.522,A 0.000,B 0.000,C 90.000,E1 273.955} C_DIS
LIN {X -0.219,Y -456.013,Z 1205.519,A 0.000,B 0.000,C 90.000,E1 273.498} C_DIS
LIN {X 0.009,Y -453.826,Z 1205.518,A 0.000,B 0.000,C 90.000,E1 273.212} C_DIS
LIN {X -0.192,Y -451.332,Z 1205.516,A 0.000,B 0.000,C 90.000,E1 272.980} C_DIS
LIN {X 0.045,Y -448.547,Z 1205.515,A 0.000,B 0.000,C 90.000,E1 272.694} C_DIS
LIN {X -0.067,Y -442.374,Z 1205.512,A 0.000,B 0.000,C 90.000,E1 272.236} C_DIS
LIN {X 0.032,Y -438.896,Z 1205.511,A 0.000,B 0.000,C 90.000,E1 272.007} C_DIS
LIN {X -0.072,Y -431.857,Z 1205.509,A 0.000,B 0.000,C 90.000,E1 271.661} C_DIS
LIN {X -0.099,Y -424.578,Z 1205.508,A 0.000,B 0.000,C 90.000,E1 271.375} C_DIS
LIN {X -0.048,Y -414.387,Z 1205.506,A 0.000,B 0.000,C 90.000,E1 271.031} C_DIS
LIN {X -0.056,Y -404.491,Z 1205.504,A 0.000,B 0.000,C 90.000,E1 270.745} C_DIS
LIN {X 0.188,Y -393.451,Z 1205.503,A 0.000,B 0.000,C 90.000,E1 270.458} C_DIS
LIN {X 0.075,Y -385.547,Z 1205.502,A 0.000,B 0.000,C 90.000,E1 270.344} C_DIS
LIN {X -0.019,Y -373.816,Z 1205.501,A 0.000,B 0.000,C 90.000,E1 270.229} C_DIS
LIN {X 0.094,Y -365.542,Z 1205.501,A 0.000,B 0.000,C 90.000,E1 270.172} C_DIS
LIN {X 0.021,Y -181.579,Z 1205.501,A 0.000,B 0.000,C 90.000,E1 270.172} C_DIS
LIN {X 0.067,Y -180.879,Z 1205.473,A 0.000,B 0.000,C 90.000,E1 265.065} C_DIS
LIN {X -0.054,Y -178.998,Z 1205.445,A 0.000,B 0.000,C 90.000,E1 260.038} C_DIS
LIN {X 0.041,Y -178.589,Z 1205.440,A 0.000,B 0.000,C 90.000,E1 259.162} C_DIS
LIN {X -0.065,Y -175.641,Z 1205.411,A 0.000,B 0.000,C 90.000,E1 254.102} C_DIS
LIN {X -0.058,Y -172.360,Z 1205.388,A 0.000,B 0.000,C 90.000,E1 249.826} C_DIS
LIN {X -0.044,Y -171.147,Z 1205.378,A 0.000,B 0.000,C 90.000,E1 248.103} C_DIS
LIN {X 0.000,Y -167.450,Z 1205.354,A 0.000,B 0.000,C 90.000,E1 243.768} C_DIS
LIN {X 0.083,Y -166.846,Z 1205.349,A 0.000,B 0.000,C 90.000,E1 242.871} C_DIS
LIN {X -0.002,Y -162.830,Z 1205.325,A 0.000,B 0.000,C 90.000,E1 238.535} C_DIS
LIN {X -0.026,Y -161.515,Z 1205.315,A 0.000,B 0.000,C 90.000,E1 236.786} C_DIS
LIN {X 0.015,Y -157.513,Z 1205.291,A 0.000,B 0.000,C 90.000,E1 232.351} C_DIS
LIN {X 0.048,Y -155.536,Z 1205.276,A 0.000,B 0.000,C 90.000,E1 229.666} C_DIS
LIN {X -0.010,Y -151.832,Z 1205.251,A 0.000,B 0.000,C 90.000,E1 225.202} C_DIS
LIN {X 0.008,Y -150.047,Z 1205.236,A 0.000,B 0.000,C 90.000,E1 222.486} C_DIS
LIN {X 0.022,Y -146.862,Z 1205.211,A 0.000,B 0.000,C 90.000,E1 217.935} C_DIS
LIN {X 0.041,Y -145.446,Z 1205.196,A 0.000,B 0.000,C 90.000,E1 215.185} C_DIS
LIN {X 0.036,Y -142.865,Z 1205.170,A 0.000,B 0.000,C 90.000,E1 210.590} C_DIS
LIN {X -0.038,Y -141.482,Z 1205.150,A 0.000,B 0.000,C 90.000,E1 206.924} C_DIS
LIN {X -0.052,Y -139.382,Z 1205.113,A 0.000,B 0.000,C 90.000,E1 200.429} C_DIS
LIN {X -0.064,Y -138.836,Z 1205.098,A 0.000,B 0.000,C 90.000,E1 197.638} C_DIS
LIN {X -0.004,Y -138.354,Z 1205.056,A 0.000,B 0.000,C 90.000,E1 190.141} C_DIS
LIN {X -0.008,Y -139.524,Z 1205.004,A 0.000,B 0.000,C 90.000,E1 180.802} C_DIS
LIN {X -0.068,Y -141.189,Z 1204.973,A 0.000,B 0.000,C 90.000,E1 175.241} C_DIS
LIN {X 0.044,Y -142.567,Z 1204.958,A 0.000,B 0.000,C 90.000,E1 172.413} C_DIS
LIN {X -0.001,Y -144.852,Z 1204.932,A 0.000,B 0.000,C 90.000,E1 167.813} C_DIS
LIN {X -0.046,Y -147.478,Z 1204.912,A 0.000,B 0.000,C 90.000,E1 164.157} C_DIS
LIN {X -0.020,Y -150.064,Z 1204.892,A 0.000,B 0.000,C 90.000,E1 160.496} C_DIS
LIN {X -0.015,Y -153.411,Z 1204.871,A 0.000,B 0.000,C 90.000,E1 156.869} C_DIS
LIN {X 0.033,Y -156.831,Z 1204.851,A 0.000,B 0.000,C 90.000,E1 153.256} C_DIS
LIN {X -0.034,Y -160.909,Z 1204.832,A 0.000,B 0.000,C 90.000,E1 149.715} C_DIS
LIN {X 0.050,Y -163.035,Z 1204.822,A 0.000,B 0.000,C 90.000,E1 147.916} C_DIS
LIN {X 0.055,Y -167.426,Z 1204.802,A 0.000,B 0.000,C 90.000,E1 144.402} C_DIS
LIN {X -0.036,Y -171.264,Z 1204.788,A 0.000,B 0.000,C 90.000,E1 141.823} C_DIS
LIN {X 0.003,Y -176.155,Z 1204.769,A 0.000,B 0.000,C 90.000,E1 138.366} C_DIS
LIN {X 0.002,Y -180.424,Z 1204.755,A 0.000,B 0.000,C 90.000,E1 135.810} C_DIS
LIN {X -0.023,Y -185.831,Z 1204.736,A 0.000,B 0.000,C 90.000,E1 132.447} C_DIS
LIN {X 0.031,Y -190.452,Z 1204.722,A 0.000,B 0.000,C 90.000,E1 129.930} C_DIS
LIN {X -0.064,Y -196.205,Z 1204.704,A 0.000,B 0.000,C 90.000,E1 126.664} C_DIS
LIN {X 0.125,Y -201.447,Z 1204.689,A 0.000,B 0.000,C 90.000,E1 123.913} C_DIS
LIN {X -0.058,Y -201.536,Z 1204.688,A 0.000,B 0.000,C 90.000,E1 123.913} C_DIS
LIN {X -0.136,Y -311.636,Z 1204.688,A 0.000,B 0.000,C 90.000,E1 123.913} C_DIS
LIN {X -0.118,Y -316.154,Z 1204.688,A 0.000,B 0.000,C 90.000,E1 123.785} C_DIS
LIN {X 0.078,Y -318.244,Z 1204.687,A 0.000,B 0.000,C 90.000,E1 123.627} C_DIS
LIN {X 0.120,Y -321.103,Z 1204.686,A 0.000,B 0.000,C 90.000,E1 123.372} C_DIS
LIN {X 0.091,Y -324.828,Z 1204.683,A 0.000,B 0.000,C 90.000,E1 122.880} C_DIS
LIN {X 0.179,Y -326.486,Z 1204.681,A 0.000,B 0.000,C 90.000,E1 122.546} C_DIS
LIN {X -0.143,Y -331.261,Z 1204.674,A 0.000,B 0.000,C 90.000,E1 121.337} C_DIS
LIN {X 0.125,Y -342.597,Z 1204.658,A 0.000,B 0.000,C 90.000,E1 118.487} C_DIS
LIN {X -0.075,Y -355.344,Z 1204.643,A 0.000,B 0.000,C 90.000,E1 115.771} C_DIS
LIN {X -0.063,Y -369.619,Z 1204.628,A 0.000,B 0.000,C 90.000,E1 113.078} C_DIS
LIN {X -0.049,Y -383.688,Z 1204.615,A 0.000,B 0.000,C 90.000,E1 110.737} C_DIS
LIN {X 0.188,Y -399.159,Z 1204.602,A 0.000,B 0.000,C 90.000,E1 108.417} C_DIS
LIN {X 0.056,Y -416.144,Z 1204.590,A 0.000,B 0.000,C 90.000,E1 106.205} C_DIS
LIN {X -0.187,Y -434.761,Z 1204.578,A 0.000,B 0.000,C 90.000,E1 104.064} C_DIS
LIN {X 0.166,Y -454.672,Z 1204.567,A 0.000,B 0.000,C 90.000,E1 101.951} C_DIS
LIN {X -0.105,Y -469.979,Z 1204.558,A 0.000,B 0.000,C 90.000,E1 100.546} C_DIS
LIN {X -0.057,Y -472.336,Z 1204.557,A 0.000,B 0.000,C 90.000,E1 100.310} C_DIS
LIN {X -0.008,Y -474.125,Z 1204.556,A 0.000,B 0.000,C 90.000,E1 100.074} C_DIS
LIN {X -0.230,Y -475.617,Z 1204.555,A 0.000,B 0.000,C 90.000,E1 99.849} C_DIS
LIN {X 0.101,Y -476.731,Z 1204.553,A 0.000,B 0.000,C 90.000,E1 99.557} C_DIS
LIN {X -0.163,Y -478.053,Z 1204.550,A 0.000,B 0.000,C 90.000,E1 99.086} C_DIS
LIN {X -0.026,Y -478.355,Z 1204.548,A 0.000,B 0.000,C 90.000,E1 98.568} C_DIS
LIN {X 0.122,Y -477.687,Z 1204.545,A 0.000,B 0.000,C 90.000,E1 98.049} C_DIS
LIN {X -0.199,Y -475.942,Z 1204.542,A 0.000,B 0.000,C 90.000,E1 97.587} C_DIS
LIN {X 0.142,Y -474.568,Z 1204.541,A 0.000,B 0.000,C 90.000,E1 97.296} C_DIS
LIN {X -0.120,Y -458.226,Z 1204.528,A 0.000,B 0.000,C 90.000,E1 95.049} C_DIS
LIN {X -0.182,Y -440.731,Z 1204.514,A 0.000,B 0.000,C 90.000,E1 92.465} C_DIS
LIN {X -0.203,Y -423.102,Z 1204.497,A 0.000,B 0.000,C 90.000,E1 89.542} C_DIS
LIN {X -0.177,Y -411.301,Z 1204.485,A 0.000,B 0.000,C 90.000,E1 87.364} C_DIS
LIN {X 0.021,Y -399.697,Z 1204.473,A 0.000,B 0.000,C 90.000,E1 85.122} C_DIS
LIN {X -0.070,Y -389.495,Z 1204.462,A 0.000,B 0.000,C 90.000,E1 83.166} C_DIS
LIN {X 0.095,Y -379.225,Z 1204.451,A 0.000,B 0.000,C 90.000,E1 81.141} C_DIS
LIN {X 0.103,Y -370.180,Z 1204.441,A 0.000,B 0.000,C 90.000,E1 79.398} C_DIS
LIN {X 0.015,Y -360.780,Z 1204.431,A 0.000,B 0.000,C 90.000,E1 77.645} C_DIS
LIN {X -0.163,Y -351.221,Z 1204.421,A 0.000,B 0.000,C 90.000,E1 75.880} C_DIS
LIN {X -0.083,Y -340.004,Z 1204.410,A 0.000,B 0.000,C 90.000,E1 73.740} C_DIS
LIN {X 0.093,Y -325.722,Z 1204.394,A 0.000,B 0.000,C 90.000,E1 70.913} C_DIS
LIN {X 0.083,Y -312.054,Z 1204.378,A 0.000,B 0.000,C 90.000,E1 68.050} C_DIS
LIN {X 0.045,Y -297.865,Z 1204.360,A 0.000,B 0.000,C 90.000,E1 64.793} C_DIS
LIN {X 0.123,Y -286.008,Z 1204.343,A 0.000,B 0.000,C 90.000,E1 61.769} C_DIS
LIN {X -0.154,Y -273.652,Z 1204.324,A 0.000,B 0.000,C 90.000,E1 58.408} C_DIS
LIN {X -0.079,Y -262.173,Z 1204.305,A 0.000,B 0.000,C 90.000,E1 54.895} C_DIS
LIN {X 0.034,Y -252.543,Z 1204.287,A 0.000,B 0.000,C 90.000,E1 51.662} C_DIS
LIN {X -0.008,Y -242.417,Z 1204.267,A 0.000,B 0.000,C 90.000,E1 48.038} C_DIS
LIN {X -0.017,Y -234.746,Z 1204.250,A 0.000,B 0.000,C 90.000,E1 45.081} C_DIS
LIN {X 0.007,Y -225.568,Z 1204.229,A 0.000,B 0.000,C 90.000,E1 41.310} C_DIS
LIN {X -0.032,Y -218.857,Z 1204.213,A 0.000,B 0.000,C 90.000,E1 38.257} C_DIS
LIN {X -0.034,Y -212.861,Z 1204.195,A 0.000,B 0.000,C 90.000,E1 35.152} C_DIS
LIN {X -0.017,Y -206.257,Z 1204.173,A 0.000,B 0.000,C 90.000,E1 31.209} C_DIS
LIN {X 0.020,Y -200.514,Z 1204.151,A 0.000,B 0.000,C 90.000,E1 27.206} C_DIS
LIN {X 0.055,Y -195.470,Z 1204.129,A 0.000,B 0.000,C 90.000,E1 23.153} C_DIS
LIN {X -0.013,Y -191.245,Z 1204.106,A 0.000,B 0.000,C 90.000,E1 19.087} C_DIS
LIN {X 0.038,Y -187.299,Z 1204.078,A 0.000,B 0.000,C 90.000,E1 14.120} C_DIS
LIN {X 0.090,Y -184.424,Z 1204.046,A 0.000,B 0.000,C 90.000,E1 8.276} C_DIS
LIN {X 0.070,Y -185.344,Z 1203.969,A 0.000,B 0.000,C 90.000,E1 354.489} C_DIS
LIN {X 0.003,Y -188.303,Z 1203.942,A 0.000,B 0.000,C 90.000,E1 349.511} C_DIS
LIN {X -0.081,Y -192.624,Z 1203.914,A 0.000,B 0.000,C 90.000,E1 344.574} C_DIS
LIN {X 0.105,Y -197.260,Z 1203.891,A 0.000,B 0.000,C 90.000,E1 340.423} C_DIS
LIN {X -0.032,Y -202.573,Z 1203.869,A 0.000,B 0.000,C 90.000,E1 336.410} C_DIS
LIN {X -0.047,Y -208.591,Z 1203.847,A 0.000,B 0.000,C 90.000,E1 332.410} C_DIS
LIN {X 0.103,Y -213.656,Z 1203.829,A 0.000,B 0.000,C 90.000,E1 329.203} C_DIS
LIN {X 0.054,Y -220.513,Z 1203.807,A 0.000,B 0.000,C 90.000,E1 325.308} C_DIS
LIN {X 0.060,Y -228.111,Z 1203.786,A 0.000,B 0.000,C 90.000,E1 321.457} C_DIS
LIN {X -0.050,Y -234.836,Z 1203.769,A 0.000,B 0.000,C 90.000,E1 318.447} C_DIS
LIN {X 0.012,Y -241.527,Z 1203.755,A 0.000,B 0.000,C 90.000,E1 315.810} C_DIS
LIN {X 0.058,Y -249.148,Z 1203.740,A 0.000,B 0.000,C 90.000,E1 313.218} C_DIS
LIN {X 0.024,Y -260.396,Z 1203.722,A 0.000,B 0.000,C 90.000,E1 309.967} C_DIS
LIN {X -0.018,Y -272.955,Z 1203.704,A 0.000,B 0.000,C 90.000,E1 306.790} C_DIS
LIN {X 0.020,Y -283.915,Z 1203.691,A 0.000,B 0.000,C 90.000,E1 304.358} C_DIS
LIN {X -0.094,Y -295.963,Z 1203.678,A 0.000,B 0.000,C 90.000,E1 302.005} C_DIS
LIN {X -0.058,Y -305.386,Z 1203.668,A 0.000,B 0.000,C 90.000,E1 300.335} C_DIS
LIN {X -0.026,Y -315.860,Z 1203.659,A 0.000,B 0.000,C 90.000,E1 298.693} C_DIS
LIN {X 0.094,Y -325.046,Z 1203.652,A 0.000,B 0.000,C 90.000,E1 297.385} C_DIS
LIN {X 0.185,Y -335.126,Z 1203.645,A 0.000,B 0.000,C 90.000,E1 296.104} C_DIS
LIN {X -0.113,Y -350.590,Z 1203.635,A 0.000,B 0.000,C 90.000,E1 294.387} C_DIS
LIN {X 0.045,Y -368.788,Z 1203.625,A 0.000,B 0.000,C 90.000,E1 292.408} C_DIS
LIN {X 0.048,Y -390.217,Z 1203.613,A 0.000,B 0.000,C 90.000,E1 290.248} C_DIS
LIN {X -0.015,Y -400.726,Z 1203.607,A 0.000,B 0.000,C 90.000,E1 289.214} C_DIS
LIN {X -0.143,Y -413.566,Z 1203.600,A 0.000,B 0.000,C 90.000,E1 287.946} C_DIS
LIN {X -0.070,Y -421.145,Z 1203.595,A 0.000,B 0.000,C 90.000,E1 287.149} C_DIS
LIN {X 0.223,Y -428.363,Z 1203.591,A 0.000,B 0.000,C 90.000,E1 286.315} C_DIS
LIN {X -0.103,Y -435.233,Z 1203.586,A 0.000,B 0.000,C 90.000,E1 285.552} C_DIS
LIN {X 0.164,Y -441.494,Z 1203.582,A 0.000,B 0.000,C 90.000,E1 284.717} C_DIS
LIN {X 0.063,Y -447.147,Z 1203.578,A 0.000,B 0.000,C 90.000,E1 283.939} C_DIS
LIN {X 0.093,Y -450.578,Z 1203.575,A 0.000,B 0.000,C 90.000,E1 283.411} C_DIS
LIN {X -0.045,Y -455.068,Z 1203.570,A 0.000,B 0.000,C 90.000,E1 282.647} C_DIS
LIN {X -0.141,Y -458.910,Z 1203.566,A 0.000,B 0.000,C 90.000,E1 281.883} C_DIS
LIN {X 0.154,Y -462.093,Z 1203.562,A 0.000,B 0.000,C 90.000,E1 281.074} C_DIS
LIN {X -0.182,Y -463.855,Z 1203.559,A 0.000,B 0.000,C 90.000,E1 280.602} C_DIS
LIN {X -0.055,Y -465.313,Z 1203.556,A 0.000,B 0.000,C 90.000,E1 280.074} C_DIS
LIN {X 0.002,Y -466.537,Z 1203.553,A 0.000,B 0.000,C 90.000,E1 279.557} C_DIS
LIN {X 0.147,Y -467.490,Z 1203.550,A 0.000,B 0.000,C 90.000,E1 279.029} C_DIS
LIN {X 0.225,Y -468.229,Z 1203.547,A 0.000,B 0.000,C 90.000,E1 278.511} C_DIS
LIN {X -0.153,Y -468.749,Z 1203.545,A 0.000,B 0.000,C 90.000,E1 278.049} C_DIS
LIN {X -0.061,Y -469.018,Z 1203.542,A 0.000,B 0.000,C 90.000,E1 277.530} C_DIS
LIN {X 0.092,Y -469.012,Z 1203.539,A 0.000,B 0.000,C 90.000,E1 277.004} C_DIS
LIN {X 0.186,Y -468.648,Z 1203.536,A 0.000,B 0.000,C 90.000,E1 276.486} C_DIS
LIN {X -0.185,Y -467.823,Z 1203.533,A 0.000,B 0.000,C 90.000,E1 276.024} C_DIS
LIN {X -0.137,Y -466.566,Z 1203.531,A 0.000,B 0.000,C 90.000,E1 275.511} C_DIS
LIN {X -0.047,Y -464.861,Z 1203.528,A 0.000,B 0.000,C 90.000,E1 274.992} C_DIS
LIN {X 0.033,Y -462.647,Z 1203.525,A 0.000,B 0.000,C 90.000,E1 274.473} C_DIS
LIN {X 0.094,Y -459.813,Z 1203.522,A 0.000,B 0.000,C 90.000,E1 273.955} C_DIS
LIN {X 0.110,Y -456.170,Z 1203.519,A 0.000,B 0.000,C 90.000,E1 273.440} C_DIS
LIN {X -0.117,Y -453.991,Z 1203.518,A 0.000,B 0.000,C 90.000,E1 273.212} C_DIS
LIN {X -0.074,Y -448.717,Z 1203.515,A 0.000,B 0.000,C 90.000,E1 272.694} C_DIS
LIN {X -0.182,Y -442.569,Z 1203.512,A 0.000,B 0.000,C 90.000,E1 272.236} C_DIS
LIN {X -0.119,Y -435.765,Z 1203.510,A 0.000,B 0.000,C 90.000,E1 271.835} C_DIS
LIN {X 0.079,Y -428.605,Z 1203.508,A 0.000,B 0.000,C 90.000,E1 271.489} C_DIS
LIN {X -0.178,Y -421.467,Z 1203.507,A 0.000,B 0.000,C 90.000,E1 271.260} C_DIS
LIN {X -0.054,Y -411.110,Z 1203.505,A 0.000,B 0.000,C 90.000,E1 270.917} C_DIS
LIN {X -0.168,Y -404.527,Z 1203.504,A 0.000,B 0.000,C 90.000,E1 270.745} C_DIS
LIN {X -0.187,Y -397.258,Z 1203.503,A 0.000,B 0.000,C 90.000,E1 270.573} C_DIS
LIN {X -0.050,Y -385.299,Z 1203.502,A 0.000,B 0.000,C 90.000,E1 270.344} C_DIS
LIN {X -0.147,Y -373.311,Z 1203.501,A 0.000,B 0.000,C 90.000,E1 270.229} C_DIS
LIN {X 0.019,Y -366.629,Z 1203.501,A 0.000,B 0.000,C 90.000,E1 270.172} C_DIS
LIN {X -0.015,Y -181.579,Z 1203.501,A 0.000,B 0.000,C 90.000,E1 270.172} C_DIS
LIN {X 0.012,Y -180.876,Z 1203.473,A 0.000,B 0.000,C 90.000,E1 265.065} C_DIS
LIN {X 0.068,Y -178.993,Z 1203.444,A 0.000,B 0.000,C 90.000,E1 259.982} C_DIS
LIN {X -0.014,Y -178.576,Z 1203.440,A 0.000,B 0.000,C 90.000,E1 259.162} C_DIS
LIN {X 0.049,Y -175.629,Z 1203.411,A 0.000,B 0.000,C 90.000,E1 254.047} C_DIS
LIN {X -0.053,Y -172.349,Z 1203.388,A 0.000,B 0.000,C 90.000,E1 249.806} C_DIS
LIN {X -0.099,Y -171.129,Z 1203.378,A 0.000,B 0.000,C 90.000,E1 248.103} C_DIS
LIN {X -0.054,Y -167.437,Z 1203.354,A 0.000,B 0.000,C 90.000,E1 243.768} C_DIS
LIN {X 0.030,Y -166.833,Z 1203.349,A 0.000,B 0.000,C 90.000,E1 242.871} C_DIS
LIN {X -0.053,Y -162.815,Z 1203.325,A 0.000,B 0.000,C 90.000,E1 238.535} C_DIS
LIN {X 0.010,Y -161.502,Z 1203.315,A 0.000,B 0.000,C 90.000,E1 236.755} C_DIS
LIN {X -0.037,Y -157.499,Z 1203.291,A 0.000,B 0.000,C 90.000,E1 232.351} C_DIS
LIN {X -0.002,Y -155.519,Z 1203.276,A 0.000,B 0.000,C 90.000,E1 229.666} C_DIS
